LIN {X 226.123,Y -181.572,Z 120.218,A 141.236,B 90.000,C 0.000} C_DIS
LIN {X 226.096,Y -181.605,Z 120.167,A 141.228,B 90.000,C 0.000} C_DIS
LIN {X 225.969,Y -181.764,Z 120.125,A 141.188,B 90.000,C 0.000} C_DIS
LIN {X 225.915,Y -181.830,Z 120.023,A 141.171,B 90.000,C 0.000} C_DIS
LIN {X 225.787,Y -181.989,Z 119.980,A 141.130,B 90.000,C 0.000} C_DIS
LIN {X 225.761,Y -182.022,Z 119.929,A 141.122,B 90.000,C 0.000} C_DIS
LIN {X 225.721,Y -182.072,Z 119.878,A 141.109,B 90.000,C 0.000} C_DIS
LIN {X 225.528,Y -182.310,Z 119.836,A 141.049,B 90.000,C 0.000} C_DIS
LIN {X 225.488,Y -182.360,Z 119.785,A 141.036,B 90.000,C 0.000} C_DIS
LIN {X 225.462,Y -182.393,Z 119.734,A 141.028,B 90.000,C 0.000} C_DIS
LIN {X 225.333,Y -182.551,Z 119.691,A 140.988,B 90.000,C 0.000} C_DIS
LIN {X 225.306,Y -182.584,Z 119.640,A 140.979,B 90.000,C 0.000} C_DIS
LIN {X 225.266,Y -182.634,Z 119.589,A 140.967,B 90.000,C 0.000} C_DIS
LIN {X 225.073,Y -182.872,Z 119.547,A 140.906,B 90.000,C 0.000} C_DIS
LIN {X 225.033,Y -182.921,Z 119.496,A 140.894,B 90.000,C 0.000} C_DIS
LIN {X 225.006,Y -182.954,Z 119.445,A 140.885,B 90.000,C 0.000} C_DIS
LIN {X 224.877,Y -183.112,Z 119.402,A 140.845,B 90.000,C 0.000} C_DIS
LIN {X 224.824,Y -183.178,Z 119.300,A 140.828,B 90.000,C 0.000} C_DIS
LIN {X 224.695,Y -183.336,Z 119.258,A 140.788,B 90.000,C 0.000} C_DIS
LIN {X 224.668,Y -183.369,Z 119.207,A 140.779,B 90.000,C 0.000} C_DIS
LIN {X 224.628,Y -183.419,Z 119.156,A 140.767,B 90.000,C 0.000} C_DIS
LIN {X 224.434,Y -183.656,Z 119.113,A 140.706,B 90.000,C 0.000} C_DIS
LIN {X 224.394,Y -183.705,Z 119.062,A 140.694,B 90.000,C 0.000} C_DIS
LIN {X 224.367,Y -183.738,Z 119.011,A 140.685,B 90.000,C 0.000} C_DIS
LIN {X 224.237,Y -183.896,Z 118.969,A 140.645,B 90.000,C 0.000} C_DIS
LIN {X 224.183,Y -183.961,Z 118.867,A 140.628,B 90.000,C 0.000} C_DIS
LIN {X 224.054,Y -184.119,Z 118.824,A 140.588,B 90.000,C 0.000} C_DIS
LIN {X 224.027,Y -184.152,Z 118.773,A 140.580,B 90.000,C 0.000} C_DIS
LIN {X 223.986,Y -184.201,Z 118.722,A 140.567,B 90.000,C 0.000} C_DIS
LIN {X 223.792,Y -184.438,Z 118.680,A 140.506,B 90.000,C 0.000} C_DIS
LIN {X 223.751,Y -184.487,Z 118.629,A 140.494,B 90.000,C 0.000} C_DIS
LIN {X 223.724,Y -184.519,Z 118.578,A 140.485,B 90.000,C 0.000} C_DIS
LIN {X 223.594,Y -184.677,Z 118.535,A 140.445,B 90.000,C 0.000} C_DIS
LIN {X 223.567,Y -184.710,Z 118.484,A 140.437,B 90.000,C 0.000} C_DIS
LIN {X 223.527,Y -184.759,Z 118.433,A 140.424,B 90.000,C 0.000} C_DIS
LIN {X 223.332,Y -184.995,Z 118.391,A 140.364,B 90.000,C 0.000} C_DIS
LIN {X 223.291,Y -185.044,Z 118.340,A 140.351,B 90.000,C 0.000} C_DIS
LIN {X 223.264,Y -185.076,Z 118.288,A 140.343,B 90.000,C 0.000} C_DIS
LIN {X 223.134,Y -185.233,Z 118.246,A 140.302,B 90.000,C 0.000} C_DIS
LIN {X 223.079,Y -185.299,Z 118.144,A 140.286,B 90.000,C 0.000} C_DIS
LIN {X 222.949,Y -185.456,Z 118.101,A 140.245,B 90.000,C 0.000} C_DIS
LIN {X 222.922,Y -185.488,Z 118.050,A 140.237,B 90.000,C 0.000} C_DIS
LIN {X 222.881,Y -185.537,Z 117.999,A 140.224,B 90.000,C 0.000} C_DIS
LIN {X 222.685,Y -185.773,Z 117.957,A 140.164,B 90.000,C 0.000} C_DIS
LIN {X 222.644,Y -185.822,Z 117.906,A 140.151,B 90.000,C 0.000} C_DIS
LIN {X 222.617,Y -185.854,Z 117.855,A 140.143,B 90.000,C 0.000} C_DIS
LIN {X 222.486,Y -186.011,Z 117.812,A 140.102,B 90.000,C 0.000} C_DIS
LIN {X 222.459,Y -186.043,Z 117.761,A 140.094,B 90.000,C 0.000} C_DIS
LIN {X 222.418,Y -186.092,Z 117.710,A 140.082,B 90.000,C 0.000} C_DIS
LIN {X 222.221,Y -186.327,Z 117.668,A 140.021,B 90.000,C 0.000} C_DIS
LIN {X 222.180,Y -186.376,Z 117.617,A 140.008,B 90.000,C 0.000} C_DIS
LIN {X 222.153,Y -186.408,Z 117.566,A 140.000,B 90.000,C 0.000} C_DIS
LIN {X 222.022,Y -186.565,Z 117.523,A 139.960,B 90.000,C 0.000} C_DIS
LIN {X 221.967,Y -186.630,Z 117.421,A 139.943,B 90.000,C 0.000} C_DIS
LIN {X 221.836,Y -186.786,Z 117.379,A 139.903,B 90.000,C 0.000} C_DIS
LIN {X 221.808,Y -186.818,Z 117.328,A 139.894,B 90.000,C 0.000} C_DIS
LIN {X 221.767,Y -186.867,Z 117.277,A 139.882,B 90.000,C 0.000} C_DIS
LIN {X 221.570,Y -187.101,Z 117.234,A 139.821,B 90.000,C 0.000} C_DIS
LIN {X 221.529,Y -187.150,Z 117.183,A 139.809,B 90.000,C 0.000} C_DIS
LIN {X 221.501,Y -187.182,Z 117.132,A 139.800,B 90.000,C 0.000} C_DIS
LIN {X 221.370,Y -187.338,Z 117.090,A 139.760,B 90.000,C 0.000} C_DIS
LIN {X 221.315,Y -187.403,Z 116.988,A 139.743,B 90.000,C 0.000} C_DIS
LIN {X 221.183,Y -187.559,Z 116.945,A 139.703,B 90.000,C 0.000} C_DIS
LIN {X 221.155,Y -187.591,Z 116.894,A 139.694,B 90.000,C 0.000} C_DIS
LIN {X 221.114,Y -187.640,Z 116.843,A 139.682,B 90.000,C 0.000} C_DIS
LIN {X 220.916,Y -187.873,Z 116.801,A 139.621,B 90.000,C 0.000} C_DIS
LIN {X 220.875,Y -187.921,Z 116.750,A 139.609,B 90.000,C 0.000} C_DIS
LIN {X 220.847,Y -187.954,Z 116.699,A 139.600,B 90.000,C 0.000} C_DIS
LIN {X 220.715,Y -188.109,Z 116.656,A 139.560,B 90.000,C 0.000} C_DIS
LIN {X 220.687,Y -188.141,Z 116.605,A 139.552,B 90.000,C 0.000} C_DIS
LIN {X 220.646,Y -188.190,Z 116.554,A 139.539,B 90.000,C 0.000} C_DIS
LIN {X 220.447,Y -188.423,Z 116.512,A 139.478,B 90.000,C 0.000} C_DIS
LIN {X 220.406,Y -188.471,Z 116.461,A 139.466,B 90.000,C 0.000} C_DIS
LIN {X 220.378,Y -188.503,Z 116.410,A 139.457,B 90.000,C 0.000} C_DIS
LIN {X 220.245,Y -188.659,Z 116.367,A 139.417,B 90.000,C 0.000} C_DIS
LIN {X 220.218,Y -188.691,Z 116.316,A 139.409,B 90.000,C 0.000} C_DIS
LIN {X 220.176,Y -188.739,Z 116.265,A 139.396,B 90.000,C 0.000} C_DIS
LIN {X 219.977,Y -188.972,Z 116.223,A 139.336,B 90.000,C 0.000} C_DIS
LIN {X 219.935,Y -189.020,Z 116.172,A 139.323,B 90.000,C 0.000} C_DIS
LIN {X 219.908,Y -189.052,Z 116.121,A 139.315,B 90.000,C 0.000} C_DIS
LIN {X 219.774,Y -189.207,Z 116.078,A 139.274,B 90.000,C 0.000} C_DIS
LIN {X 219.719,Y -189.271,Z 115.976,A 139.258,B 90.000,C 0.000} C_DIS
LIN {X 219.586,Y -189.426,Z 115.934,A 139.217,B 90.000,C 0.000} C_DIS
LIN {X 219.558,Y -189.458,Z 115.883,A 139.209,B 90.000,C 0.000} C_DIS
LIN {X 219.516,Y -189.506,Z 115.831,A 139.196,B 90.000,C 0.000} C_DIS
LIN {X 219.316,Y -189.738,Z 115.789,A 139.136,B 90.000,C 0.000} C_DIS
LIN {X 219.274,Y -189.786,Z 115.738,A 139.123,B 90.000,C 0.000} C_DIS
LIN {X 219.247,Y -189.818,Z 115.687,A 139.115,B 90.000,C 0.000} C_DIS
LIN {X 219.113,Y -189.972,Z 115.645,A 139.075,B 90.000,C 0.000} C_DIS
LIN {X 219.057,Y -190.036,Z 115.542,A 139.058,B 90.000,C 0.000} C_DIS
LIN {X 218.924,Y -190.191,Z 115.500,A 139.017,B 90.000,C 0.000} C_DIS
LIN {X 218.896,Y -190.223,Z 115.449,A 139.009,B 90.000,C 0.000} C_DIS
LIN {X 218.854,Y -190.271,Z 115.398,A 138.996,B 90.000,C 0.000} C_DIS
LIN {X 218.653,Y -190.502,Z 115.355,A 138.936,B 90.000,C 0.000} C_DIS
LIN {X 218.611,Y -190.550,Z 115.304,A 138.923,B 90.000,C 0.000} C_DIS
LIN {X 218.583,Y -190.582,Z 115.253,A 138.915,B 90.000,C 0.000} C_DIS
LIN {X 218.449,Y -190.736,Z 115.211,A 138.875,B 90.000,C 0.000} C_DIS
LIN {X 218.421,Y -190.768,Z 115.160,A 138.866,B 90.000,C 0.000} C_DIS
LIN {X 218.379,Y -190.816,Z 115.109,A 138.854,B 90.000,C 0.000} C_DIS
LIN {X 218.178,Y -191.046,Z 115.066,A 138.793,B 90.000,C 0.000} C_DIS
LIN {X 218.136,Y -191.094,Z 115.015,A 138.781,B 90.000,C 0.000} C_DIS
LIN {X 218.108,Y -191.126,Z 114.964,A 138.772,B 90.000,C 0.000} C_DIS
LIN {X 217.973,Y -191.279,Z 114.922,A 138.732,B 90.000,C 0.000} C_DIS
LIN {X 217.917,Y -191.343,Z 114.820,A 138.715,B 90.000,C 0.000} C_DIS
LIN {X 217.782,Y -191.497,Z 114.777,A 138.675,B 90.000,C 0.000} C_DIS
LIN {X 217.754,Y -191.528,Z 114.726,A 138.666,B 90.000,C 0.000} C_DIS
LIN {X 217.712,Y -191.576,Z 114.675,A 138.654,B 90.000,C 0.000} C_DIS
LIN {X 217.510,Y -191.806,Z 114.633,A 138.593,B 90.000,C 0.000} C_DIS
LIN {X 217.468,Y -191.854,Z 114.582,A 138.581,B 90.000,C 0.000} C_DIS
LIN {X 217.439,Y -191.886,Z 114.531,A 138.572,B 90.000,C 0.000} C_DIS
LIN {X 217.304,Y -192.039,Z 114.488,A 138.532,B 90.000,C 0.000} C_DIS
LIN {X 217.248,Y -192.102,Z 114.386,A 138.515,B 90.000,C 0.000} C_DIS
LIN {X 217.113,Y -192.255,Z 114.344,A 138.475,B 90.000,C 0.000} C_DIS
LIN {X 217.085,Y -192.287,Z 114.293,A 138.466,B 90.000,C 0.000} C_DIS
LIN {X 217.042,Y -192.335,Z 114.242,A 138.454,B 90.000,C 0.000} C_DIS
LIN {X 216.839,Y -192.564,Z 114.199,A 138.393,B 90.000,C 0.000} C_DIS
LIN {X 216.797,Y -192.611,Z 114.148,A 138.381,B 90.000,C 0.000} C_DIS
LIN {X 216.769,Y -192.643,Z 114.097,A 138.372,B 90.000,C 0.000} C_DIS
LIN {X 216.633,Y -192.796,Z 114.055,A 138.332,B 90.000,C 0.000} C_DIS
LIN {X 216.605,Y -192.827,Z 114.004,A 138.324,B 90.000,C 0.000} C_DIS
LIN {X 216.563,Y -192.875,Z 113.953,A 138.311,B 90.000,C 0.000} C_DIS
LIN {X 216.359,Y -193.103,Z 113.910,A 138.251,B 90.000,C 0.000} C_DIS
LIN {X 216.316,Y -193.151,Z 113.859,A 138.238,B 90.000,C 0.000} C_DIS
LIN {X 216.288,Y -193.183,Z 113.808,A 138.230,B 90.000,C 0.000} C_DIS
LIN {X 216.152,Y -193.335,Z 113.766,A 138.189,B 90.000,C 0.000} C_DIS
LIN {X 216.095,Y -193.398,Z 113.664,A 138.173,B 90.000,C 0.000} C_DIS
LIN {X 215.959,Y -193.550,Z 113.621,A 138.132,B 90.000,C 0.000} C_DIS
LIN {X 215.931,Y -193.582,Z 113.570,A 138.124,B 90.000,C 0.000} C_DIS
LIN {X 215.888,Y -193.629,Z 113.519,A 138.111,B 90.000,C 0.000} C_DIS
LIN {X 215.684,Y -193.857,Z 113.477,A 138.051,B 90.000,C 0.000} C_DIS
LIN {X 215.641,Y -193.904,Z 113.426,A 138.038,B 90.000,C 0.000} C_DIS
LIN {X 215.613,Y -193.936,Z 113.375,A 138.030,B 90.000,C 0.000} C_DIS
LIN {X 215.476,Y -194.088,Z 113.332,A 137.989,B 90.000,C 0.000} C_DIS
LIN {X 215.448,Y -194.119,Z 113.281,A 137.981,B 90.000,C 0.000} C_DIS
LIN {X 215.405,Y -194.166,Z 113.230,A 137.968,B 90.000,C 0.000} C_DIS
LIN {X 215.200,Y -194.394,Z 113.188,A 137.908,B 90.000,C 0.000} C_DIS
LIN {X 215.157,Y -194.441,Z 113.137,A 137.895,B 90.000,C 0.000} C_DIS
LIN {X 215.129,Y -194.473,Z 113.085,A 137.887,B 90.000,C 0.000} C_DIS
LIN {X 214.992,Y -194.624,Z 113.043,A 137.847,B 90.000,C 0.000} C_DIS
LIN {X 214.935,Y -194.687,Z 112.941,A 137.830,B 90.000,C 0.000} C_DIS
LIN {X 214.798,Y -194.838,Z 112.898,A 137.790,B 90.000,C 0.000} C_DIS
LIN {X 214.769,Y -194.870,Z 112.847,A 137.781,B 90.000,C 0.000} C_DIS
LIN {X 214.726,Y -194.917,Z 112.796,A 137.769,B 90.000,C 0.000} C_DIS
LIN {X 214.521,Y -195.143,Z 112.754,A 137.708,B 90.000,C 0.000} C_DIS
LIN {X 214.478,Y -195.190,Z 112.703,A 137.695,B 90.000,C 0.000} C_DIS
LIN {X 214.449,Y -195.222,Z 112.652,A 137.687,B 90.000,C 0.000} C_DIS
LIN {X 214.312,Y -195.373,Z 112.609,A 137.647,B 90.000,C 0.000} C_DIS
LIN {X 214.254,Y -195.436,Z 112.507,A 137.630,B 90.000,C 0.000} C_DIS
LIN {X 214.117,Y -195.586,Z 112.465,A 137.590,B 90.000,C 0.000} C_DIS
LIN {X 214.088,Y -195.618,Z 112.414,A 137.581,B 90.000,C 0.000} C_DIS
LIN {X 214.045,Y -195.665,Z 112.363,A 137.569,B 90.000,C 0.000} C_DIS
LIN {X 213.838,Y -195.891,Z 112.320,A 137.508,B 90.000,C 0.000} C_DIS
LIN {X 213.795,Y -195.938,Z 112.269,A 137.496,B 90.000,C 0.000} C_DIS
LIN {X 213.767,Y -195.969,Z 112.218,A 137.487,B 90.000,C 0.000} C_DIS
LIN {X 213.629,Y -196.119,Z 112.176,A 137.447,B 90.000,C 0.000} C_DIS
LIN {X 213.600,Y -196.151,Z 112.125,A 137.439,B 90.000,C 0.000} C_DIS
LIN {X 213.557,Y -196.197,Z 112.074,A 137.426,B 90.000,C 0.000} C_DIS
LIN {X 213.350,Y -196.423,Z 112.031,A 137.365,B 90.000,C 0.000} C_DIS
LIN {X 213.307,Y -196.470,Z 111.980,A 137.353,B 90.000,C 0.000} C_DIS
LIN {X 213.278,Y -196.501,Z 111.929,A 137.344,B 90.000,C 0.000} C_DIS
LIN {X 213.139,Y -196.651,Z 111.887,A 137.304,B 90.000,C 0.000} C_DIS
LIN {X 213.111,Y -196.682,Z 111.836,A 137.296,B 90.000,C 0.000} C_DIS
LIN {X 213.067,Y -196.729,Z 111.785,A 137.283,B 90.000,C 0.000} C_DIS
LIN {X 212.860,Y -196.954,Z 111.742,A 137.223,B 90.000,C 0.000} C_DIS
LIN {X 212.816,Y -197.001,Z 111.691,A 137.210,B 90.000,C 0.000} C_DIS
LIN {X 212.787,Y -197.032,Z 111.640,A 137.202,B 90.000,C 0.000} C_DIS
LIN {X 212.649,Y -197.181,Z 111.598,A 137.161,B 90.000,C 0.000} C_DIS
LIN {X 212.591,Y -197.244,Z 111.496,A 137.145,B 90.000,C 0.000} C_DIS
LIN {X 212.452,Y -197.393,Z 111.453,A 137.104,B 90.000,C 0.000} C_DIS
LIN {X 212.423,Y -197.424,Z 111.402,A 137.096,B 90.000,C 0.000} C_DIS
LIN {X 212.380,Y -197.471,Z 111.351,A 137.083,B 90.000,C 0.000} C_DIS
LIN {X 212.171,Y -197.695,Z 111.309,A 137.023,B 90.000,C 0.000} C_DIS
LIN {X 212.128,Y -197.742,Z 111.258,A 137.010,B 90.000,C 0.000} C_DIS
LIN {X 212.099,Y -197.773,Z 111.207,A 137.002,B 90.000,C 0.000} C_DIS
LIN {X 211.959,Y -197.922,Z 111.164,A 136.961,B 90.000,C 0.000} C_DIS
LIN {X 211.902,Y -197.984,Z 111.062,A 136.945,B 90.000,C 0.000} C_DIS
LIN {X 211.762,Y -198.133,Z 111.020,A 136.904,B 90.000,C 0.000} C_DIS
LIN {X 211.733,Y -198.164,Z 110.969,A 136.896,B 90.000,C 0.000} C_DIS
LIN {X 211.690,Y -198.211,Z 110.918,A 136.883,B 90.000,C 0.000} C_DIS
LIN {X 211.480,Y -198.434,Z 110.875,A 136.823,B 90.000,C 0.000} C_DIS
LIN {X 211.437,Y -198.481,Z 110.824,A 136.810,B 90.000,C 0.000} C_DIS
LIN {X 211.408,Y -198.512,Z 110.773,A 136.802,B 90.000,C 0.000} C_DIS
LIN {X 211.268,Y -198.660,Z 110.731,A 136.762,B 90.000,C 0.000} C_DIS
LIN {X 211.239,Y -198.691,Z 110.680,A 136.753,B 90.000,C 0.000} C_DIS
LIN {X 211.195,Y -198.738,Z 110.628,A 136.741,B 90.000,C 0.000} C_DIS
LIN {X 210.985,Y -198.961,Z 110.586,A 136.680,B 90.000,C 0.000} C_DIS
LIN {X 210.941,Y -199.007,Z 110.535,A 136.668,B 90.000,C 0.000} C_DIS
LIN {X 210.912,Y -199.038,Z 110.484,A 136.659,B 90.000,C 0.000} C_DIS
LIN {X 210.772,Y -199.186,Z 110.442,A 136.619,B 90.000,C 0.000} C_DIS
LIN {X 210.714,Y -199.248,Z 110.339,A 136.602,B 90.000,C 0.000} C_DIS
LIN {X 210.573,Y -199.396,Z 110.297,A 136.562,B 90.000,C 0.000} C_DIS
LIN {X 210.544,Y -199.427,Z 110.246,A 136.553,B 90.000,C 0.000} C_DIS
LIN {X 210.500,Y -199.473,Z 110.195,A 136.541,B 90.000,C 0.000} C_DIS
LIN {X 210.290,Y -199.695,Z 110.152,A 136.480,B 90.000,C 0.000} C_DIS
LIN {X 210.246,Y -199.742,Z 110.101,A 136.468,B 90.000,C 0.000} C_DIS
LIN {X 210.217,Y -199.772,Z 110.050,A 136.459,B 90.000,C 0.000} C_DIS
LIN {X 210.076,Y -199.920,Z 110.008,A 136.419,B 90.000,C 0.000} C_DIS
LIN {X 210.017,Y -199.982,Z 109.906,A 136.402,B 90.000,C 0.000} C_DIS
LIN {X 209.877,Y -200.130,Z 109.863,A 136.362,B 90.000,C 0.000} C_DIS
LIN {X 209.847,Y -200.160,Z 109.812,A 136.353,B 90.000,C 0.000} C_DIS
LIN {X 209.803,Y -200.206,Z 109.761,A 136.341,B 90.000,C 0.000} C_DIS
LIN {X 209.592,Y -200.428,Z 109.719,A 136.280,B 90.000,C 0.000} C_DIS
LIN {X 209.548,Y -200.474,Z 109.668,A 136.268,B 90.000,C 0.000} C_DIS
LIN {X 209.518,Y -200.505,Z 109.617,A 136.259,B 90.000,C 0.000} C_DIS
LIN {X 209.377,Y -200.652,Z 109.574,A 136.219,B 90.000,C 0.000} C_DIS
LIN {X 209.348,Y -200.683,Z 109.523,A 136.211,B 90.000,C 0.000} C_DIS
LIN {X 209.304,Y -200.729,Z 109.472,A 136.198,B 90.000,C 0.000} C_DIS
LIN {X 209.092,Y -200.949,Z 109.430,A 136.138,B 90.000,C 0.000} C_DIS
LIN {X 209.048,Y -200.995,Z 109.379,A 136.125,B 90.000,C 0.000} C_DIS
LIN {X 209.018,Y -201.026,Z 109.328,A 136.117,B 90.000,C 0.000} C_DIS
LIN {X 208.877,Y -201.173,Z 109.285,A 136.076,B 90.000,C 0.000} C_DIS
LIN {X 208.818,Y -201.234,Z 109.183,A 136.059,B 90.000,C 0.000} C_DIS
LIN {X 208.676,Y -201.381,Z 109.141,A 136.019,B 90.000,C 0.000} C_DIS
LIN {X 208.646,Y -201.412,Z 109.090,A 136.011,B 90.000,C 0.000} C_DIS
LIN {X 208.602,Y -201.458,Z 109.039,A 135.998,B 90.000,C 0.000} C_DIS
LIN {X 208.389,Y -201.678,Z 108.996,A 135.938,B 90.000,C 0.000} C_DIS
LIN {X 208.345,Y -201.723,Z 108.945,A 135.925,B 90.000,C 0.000} C_DIS
LIN {X 208.316,Y -201.754,Z 108.894,A 135.917,B 90.000,C 0.000} C_DIS
LIN {X 208.173,Y -201.901,Z 108.852,A 135.876,B 90.000,C 0.000} C_DIS
LIN {X 208.144,Y -201.931,Z 108.801,A 135.868,B 90.000,C 0.000} C_DIS
LIN {X 208.100,Y -201.977,Z 108.750,A 135.855,B 90.000,C 0.000} C_DIS
LIN {X 207.886,Y -202.196,Z 108.707,A 135.795,B 90.000,C 0.000} C_DIS
LIN {X 207.842,Y -202.242,Z 108.656,A 135.782,B 90.000,C 0.000} C_DIS
LIN {X 207.812,Y -202.272,Z 108.605,A 135.774,B 90.000,C 0.000} C_DIS
LIN {X 207.670,Y -202.419,Z 108.563,A 135.734,B 90.000,C 0.000} C_DIS
LIN {X 207.610,Y -202.479,Z 108.461,A 135.717,B 90.000,C 0.000} C_DIS
LIN {X 207.468,Y -202.626,Z 108.418,A 135.677,B 90.000,C 0.000} C_DIS
LIN {X 207.438,Y -202.656,Z 108.367,A 135.668,B 90.000,C 0.000} C_DIS
LIN {X 207.394,Y -202.701,Z 108.316,A 135.656,B 90.000,C 0.000} C_DIS
LIN {X 207.179,Y -202.920,Z 108.274,A 135.595,B 90.000,C 0.000} C_DIS
LIN {X 207.135,Y -202.966,Z 108.223,A 135.582,B 90.000,C 0.000} C_DIS
LIN {X 207.105,Y -202.996,Z 108.172,A 135.574,B 90.000,C 0.000} C_DIS
LIN {X 206.962,Y -203.142,Z 108.129,A 135.534,B 90.000,C 0.000} C_DIS
LIN {X 206.933,Y -203.172,Z 108.078,A 135.525,B 90.000,C 0.000} C_DIS
LIN {X 206.888,Y -203.218,Z 108.027,A 135.513,B 90.000,C 0.000} C_DIS
LIN {X 206.673,Y -203.436,Z 107.985,A 135.452,B 90.000,C 0.000} C_DIS
LIN {X 206.629,Y -203.481,Z 107.933,A 135.440,B 90.000,C 0.000} C_DIS
LIN {X 206.599,Y -203.512,Z 107.882,A 135.431,B 90.000,C 0.000} C_DIS
LIN {X 206.455,Y -203.657,Z 107.840,A 135.391,B 90.000,C 0.000} C_DIS
LIN {X 206.396,Y -203.717,Z 107.738,A 135.374,B 90.000,C 0.000} C_DIS
LIN {X 206.252,Y -203.863,Z 107.695,A 135.334,B 90.000,C 0.000} C_DIS
LIN {X 206.222,Y -203.893,Z 107.644,A 135.325,B 90.000,C 0.000} C_DIS
LIN {X 206.178,Y -203.938,Z 107.593,A 135.313,B 90.000,C 0.000} C_DIS
LIN {X 205.962,Y -204.156,Z 107.551,A 135.252,B 90.000,C 0.000} C_DIS
LIN {X 205.917,Y -204.201,Z 107.500,A 135.240,B 90.000,C 0.000} C_DIS
LIN {X 205.887,Y -204.231,Z 107.449,A 135.231,B 90.000,C 0.000} C_DIS
LIN {X 205.744,Y -204.376,Z 107.406,A 135.191,B 90.000,C 0.000} C_DIS
LIN {X 205.684,Y -204.436,Z 107.304,A 135.174,B 90.000,C 0.000} C_DIS
LIN {X 205.540,Y -204.581,Z 107.262,A 135.134,B 90.000,C 0.000} C_DIS
LIN {X 205.510,Y -204.611,Z 107.211,A 135.126,B 90.000,C 0.000} C_DIS
LIN {X 205.465,Y -204.656,Z 107.160,A 135.113,B 90.000,C 0.000} C_DIS
LIN {X 205.249,Y -204.873,Z 107.117,A 135.052,B 90.000,C 0.000} C_DIS
LIN {X 205.204,Y -204.918,Z 107.066,A 135.040,B 90.000,C 0.000} C_DIS
LIN {X 205.174,Y -204.948,Z 107.015,A 135.032,B 90.000,C 0.000} C_DIS
LIN {X 205.029,Y -205.093,Z 106.973,A 134.991,B 90.000,C 0.000} C_DIS
LIN {X 204.999,Y -205.123,Z 106.922,A 134.983,B 90.000,C 0.000} C_DIS
LIN {X 204.954,Y -205.168,Z 106.871,A 134.970,B 90.000,C 0.000} C_DIS
LIN {X 204.738,Y -205.384,Z 106.828,A 134.910,B 90.000,C 0.000} C_DIS
LIN {X 204.692,Y -205.429,Z 106.777,A 134.897,B 90.000,C 0.000} C_DIS
LIN {X 204.662,Y -205.459,Z 106.726,A 134.889,B 90.000,C 0.000} C_DIS
LIN {X 204.518,Y -205.603,Z 106.684,A 134.848,B 90.000,C 0.000} C_DIS
LIN {X 204.458,Y -205.663,Z 106.582,A 134.832,B 90.000,C 0.000} C_DIS
LIN {X 204.313,Y -205.807,Z 106.539,A 134.791,B 90.000,C 0.000} C_DIS
LIN {X 204.283,Y -205.836,Z 106.488,A 134.783,B 90.000,C 0.000} C_DIS
LIN {X 204.237,Y -205.881,Z 106.437,A 134.770,B 90.000,C 0.000} C_DIS
LIN {X 204.020,Y -206.097,Z 106.395,A 134.710,B 90.000,C 0.000} C_DIS
LIN {X 203.975,Y -206.142,Z 106.344,A 134.697,B 90.000,C 0.000} C_DIS
LIN {X 203.944,Y -206.171,Z 106.293,A 134.689,B 90.000,C 0.000} C_DIS
LIN {X 203.799,Y -206.315,Z 106.250,A 134.649,B 90.000,C 0.000} C_DIS
LIN {X 203.769,Y -206.345,Z 106.199,A 134.640,B 90.000,C 0.000} C_DIS
LIN {X 203.724,Y -206.390,Z 106.148,A 134.628,B 90.000,C 0.000} C_DIS
LIN {X 203.506,Y -206.605,Z 106.106,A 134.567,B 90.000,C 0.000} C_DIS
LIN {X 203.460,Y -206.649,Z 106.055,A 134.554,B 90.000,C 0.000} C_DIS
LIN {X 203.430,Y -206.679,Z 106.004,A 134.546,B 90.000,C 0.000} C_DIS
LIN {X 203.284,Y -206.822,Z 105.961,A 134.506,B 90.000,C 0.000} C_DIS
LIN {X 203.224,Y -206.882,Z 105.859,A 134.489,B 90.000,C 0.000} C_DIS
LIN {X 203.078,Y -207.025,Z 105.817,A 134.449,B 90.000,C 0.000} C_DIS
LIN {X 203.048,Y -207.054,Z 105.766,A 134.440,B 90.000,C 0.000} C_DIS
LIN {X 203.002,Y -207.099,Z 105.715,A 134.428,B 90.000,C 0.000} C_DIS
LIN {X 202.784,Y -207.313,Z 105.672,A 134.367,B 90.000,C 0.000} C_DIS
LIN {X 202.738,Y -207.358,Z 105.621,A 134.355,B 90.000,C 0.000} C_DIS
LIN {X 202.708,Y -207.387,Z 105.570,A 134.346,B 90.000,C 0.000} C_DIS
LIN {X 202.562,Y -207.530,Z 105.528,A 134.306,B 90.000,C 0.000} C_DIS
LIN {X 202.531,Y -207.560,Z 105.477,A 134.297,B 90.000,C 0.000} C_DIS
LIN {X 202.486,Y -207.604,Z 105.425,A 134.285,B 90.000,C 0.000} C_DIS
LIN {X 202.266,Y -207.818,Z 105.383,A 134.224,B 90.000,C 0.000} C_DIS
LIN {X 202.221,Y -207.862,Z 105.332,A 134.212,B 90.000,C 0.000} C_DIS
LIN {X 202.190,Y -207.892,Z 105.281,A 134.203,B 90.000,C 0.000} C_DIS
LIN {X 202.044,Y -208.034,Z 105.238,A 134.163,B 90.000,C 0.000} C_DIS
LIN {X 201.983,Y -208.093,Z 105.136,A 134.146,B 90.000,C 0.000} C_DIS
LIN {X 201.836,Y -208.236,Z 105.094,A 134.106,B 90.000,C 0.000} C_DIS
LIN {X 201.806,Y -208.265,Z 105.043,A 134.098,B 90.000,C 0.000} C_DIS
LIN {X 201.760,Y -208.309,Z 104.992,A 134.085,B 90.000,C 0.000} C_DIS
LIN {X 201.540,Y -208.522,Z 104.949,A 134.025,B 90.000,C 0.000} C_DIS
LIN {X 201.494,Y -208.567,Z 104.898,A 134.012,B 90.000,C 0.000} C_DIS
LIN {X 201.464,Y -208.596,Z 104.847,A 134.004,B 90.000,C 0.000} C_DIS
LIN {X 201.317,Y -208.738,Z 104.805,A 133.963,B 90.000,C 0.000} C_DIS
LIN {X 201.286,Y -208.767,Z 104.754,A 133.955,B 90.000,C 0.000} C_DIS
LIN {X 201.241,Y -208.811,Z 104.703,A 133.942,B 90.000,C 0.000} C_DIS
LIN {X 201.020,Y -209.024,Z 104.660,A 133.882,B 90.000,C 0.000} C_DIS
LIN {X 200.974,Y -209.068,Z 104.609,A 133.869,B 90.000,C 0.000} C_DIS
LIN {X 200.943,Y -209.097,Z 104.558,A 133.861,B 90.000,C 0.000} C_DIS
LIN {X 200.796,Y -209.239,Z 104.516,A 133.820,B 90.000,C 0.000} C_DIS
LIN {X 200.735,Y -209.298,Z 104.414,A 133.804,B 90.000,C 0.000} C_DIS
LIN {X 200.588,Y -209.439,Z 104.371,A 133.763,B 90.000,C 0.000} C_DIS
LIN {X 200.557,Y -209.468,Z 104.320,A 133.755,B 90.000,C 0.000} C_DIS
LIN {X 200.511,Y -209.512,Z 104.269,A 133.742,B 90.000,C 0.000} C_DIS
LIN {X 200.290,Y -209.724,Z 104.227,A 133.682,B 90.000,C 0.000} C_DIS
LIN {X 200.243,Y -209.768,Z 104.176,A 133.669,B 90.000,C 0.000} C_DIS
LIN {X 200.213,Y -209.797,Z 104.125,A 133.661,B 90.000,C 0.000} C_DIS
LIN {X 200.065,Y -209.938,Z 104.082,A 133.621,B 90.000,C 0.000} C_DIS
LIN {X 200.004,Y -209.997,Z 103.980,A 133.604,B 90.000,C 0.000} C_DIS
LIN {X 199.856,Y -210.137,Z 103.938,A 133.563,B 90.000,C 0.000} C_DIS
LIN {X 199.825,Y -210.167,Z 103.887,A 133.555,B 90.000,C 0.000} C_DIS
LIN {X 199.779,Y -210.210,Z 103.836,A 133.542,B 90.000,C 0.000} C_DIS
LIN {X 199.557,Y -210.421,Z 103.793,A 133.482,B 90.000,C 0.000} C_DIS
LIN {X 199.510,Y -210.465,Z 103.742,A 133.469,B 90.000,C 0.000} C_DIS
LIN {X 199.480,Y -210.494,Z 103.691,A 133.461,B 90.000,C 0.000} C_DIS
LIN {X 199.331,Y -210.635,Z 103.649,A 133.421,B 90.000,C 0.000} C_DIS
LIN {X 199.301,Y -210.664,Z 103.598,A 133.412,B 90.000,C 0.000} C_DIS
LIN {X 199.254,Y -210.708,Z 103.547,A 133.400,B 90.000,C 0.000} C_DIS
LIN {X 199.032,Y -210.918,Z 103.504,A 133.339,B 90.000,C 0.000} C_DIS
LIN {X 198.985,Y -210.962,Z 103.453,A 133.327,B 90.000,C 0.000} C_DIS
LIN {X 198.955,Y -210.991,Z 103.402,A 133.318,B 90.000,C 0.000} C_DIS
LIN {X 198.806,Y -211.131,Z 103.360,A 133.278,B 90.000,C 0.000} C_DIS
LIN {X 198.744,Y -211.189,Z 103.258,A 133.261,B 90.000,C 0.000} C_DIS
LIN {X 198.595,Y -211.329,Z 103.215,A 133.221,B 90.000,C 0.000} C_DIS
LIN {X 198.564,Y -211.358,Z 103.164,A 133.212,B 90.000,C 0.000} C_DIS
LIN {X 198.518,Y -211.401,Z 103.113,A 133.200,B 90.000,C 0.000} C_DIS
LIN {X 198.295,Y -211.611,Z 103.071,A 133.139,B 90.000,C 0.000} C_DIS
LIN {X 198.248,Y -211.655,Z 103.020,A 133.127,B 90.000,C 0.000} C_DIS
LIN {X 198.217,Y -211.684,Z 102.968,A 133.118,B 90.000,C 0.000} C_DIS
LIN {X 198.068,Y -211.823,Z 102.926,A 133.078,B 90.000,C 0.000} C_DIS
LIN {X 198.037,Y -211.852,Z 102.875,A 133.070,B 90.000,C 0.000} C_DIS
LIN {X 197.991,Y -211.896,Z 102.824,A 133.057,B 90.000,C 0.000} C_DIS
LIN {X 197.767,Y -212.104,Z 102.782,A 132.997,B 90.000,C 0.000} C_DIS
LIN {X 197.720,Y -212.148,Z 102.730,A 132.984,B 90.000,C 0.000} C_DIS
LIN {X 197.689,Y -212.177,Z 102.679,A 132.976,B 90.000,C 0.000} C_DIS
LIN {X 197.540,Y -212.316,Z 102.637,A 132.935,B 90.000,C 0.000} C_DIS
LIN {X 197.478,Y -212.374,Z 102.535,A 132.918,B 90.000,C 0.000} C_DIS
LIN {X 197.328,Y -212.513,Z 102.492,A 132.878,B 90.000,C 0.000} C_DIS
LIN {X 197.297,Y -212.542,Z 102.441,A 132.870,B 90.000,C 0.000} C_DIS
LIN {X 197.273,Y -212.564,Z 102.390,A 132.863,B 90.000,C 0.000} C_DIS
LIN {X 197.215,Y -212.618,Z 102.369,A 132.848,B 90.000,C 0.000} C_DIS
LIN {X 197.119,Y -212.707,Z 102.317,A 132.822,B 90.000,C 0.000} C_DIS
LIN {X 197.003,Y -212.814,Z 102.192,A 132.791,B 90.000,C 0.000} C_DIS
LIN {X 196.873,Y -212.935,Z 102.014,A 132.756,B 90.000,C 0.000} C_DIS
LIN {X 196.882,Y -212.926,Z 99.514,A 132.758,B 90.000,C 0.000} C_DIS
LIN {X 196.887,Y -212.922,Z 99.055,A 132.759,B 90.000,C 0.000} C_DIS
LIN {X 196.965,Y -212.849,Z 98.268,A 132.780,B 90.000,C 0.000} C_DIS
LIN {X 196.993,Y -212.823,Z 96.353,A 132.788,B 90.000,C 0.000} C_DIS
LIN {X 197.032,Y -212.787,Z 96.010,A 132.798,B 90.000,C 0.000} C_DIS
LIN {X 197.069,Y -212.753,Z 95.977,A 132.808,B 90.000,C 0.000} C_DIS
LIN {X 197.085,Y -212.738,Z 95.898,A 132.813,B 90.000,C 0.000} C_DIS
LIN {X 197.123,Y -212.703,Z 95.767,A 132.823,B 90.000,C 0.000} C_DIS
LIN {X 197.215,Y -212.618,Z 95.609,A 132.848,B 90.000,C 0.000} C_DIS
LIN {X 197.368,Y -212.475,Z 95.469,A 132.889,B 90.000,C 0.000} C_DIS
LIN {X 197.586,Y -212.273,Z 95.432,A 132.948,B 90.000,C 0.000} C_DIS
LIN {X 197.755,Y -212.115,Z 95.453,A 132.993,B 90.000,C 0.000} C_DIS
LIN {X 197.826,Y -212.049,Z 95.504,A 133.013,B 90.000,C 0.000} C_DIS
LIN {X 197.872,Y -212.006,Z 95.555,A 133.025,B 90.000,C 0.000} C_DIS
LIN {X 198.096,Y -211.797,Z 95.597,A 133.086,B 90.000,C 0.000} C_DIS
LIN {X 198.189,Y -211.710,Z 95.700,A 133.111,B 90.000,C 0.000} C_DIS
LIN {X 198.413,Y -211.500,Z 95.742,A 133.171,B 90.000,C 0.000} C_DIS
LIN {X 198.459,Y -211.457,Z 95.793,A 133.184,B 90.000,C 0.000} C_DIS
LIN {X 198.490,Y -211.428,Z 95.844,A 133.192,B 90.000,C 0.000} C_DIS
LIN {X 198.639,Y -211.288,Z 95.887,A 133.233,B 90.000,C 0.000} C_DIS
LIN {X 198.701,Y -211.230,Z 95.989,A 133.249,B 90.000,C 0.000} C_DIS
LIN {X 198.775,Y -211.160,Z 96.010,A 133.270,B 90.000,C 0.000} C_DIS
LIN {X 198.849,Y -211.090,Z 95.989,A 133.290,B 90.000,C 0.000} C_DIS
LIN {X 198.880,Y -211.061,Z 95.938,A 133.298,B 90.000,C 0.000} C_DIS
LIN {X 198.849,Y -211.090,Z 95.887,A 133.290,B 90.000,C 0.000} C_DIS
LIN {X 198.701,Y -211.230,Z 95.844,A 133.249,B 90.000,C 0.000} C_DIS
LIN {X 198.639,Y -211.288,Z 95.742,A 133.233,B 90.000,C 0.000} C_DIS
LIN {X 198.490,Y -211.428,Z 95.700,A 133.192,B 90.000,C 0.000} C_DIS
LIN {X 198.428,Y -211.486,Z 95.597,A 133.175,B 90.000,C 0.000} C_DIS
LIN {X 198.279,Y -211.626,Z 95.555,A 133.135,B 90.000,C 0.000} C_DIS
LIN {X 198.217,Y -211.684,Z 95.453,A 133.118,B 90.000,C 0.000} C_DIS
LIN {X 198.068,Y -211.823,Z 95.411,A 133.078,B 90.000,C 0.000} C_DIS
LIN {X 198.006,Y -211.881,Z 95.308,A 133.061,B 90.000,C 0.000} C_DIS
LIN {X 197.857,Y -212.020,Z 95.266,A 133.021,B 90.000,C 0.000} C_DIS
LIN {X 197.795,Y -212.078,Z 95.164,A 133.004,B 90.000,C 0.000} C_DIS
LIN {X 197.645,Y -212.217,Z 95.121,A 132.964,B 90.000,C 0.000} C_DIS
LIN {X 197.614,Y -212.246,Z 95.070,A 132.955,B 90.000,C 0.000} C_DIS
LIN {X 197.568,Y -212.290,Z 95.019,A 132.943,B 90.000,C 0.000} C_DIS
LIN {X 197.344,Y -212.498,Z 94.977,A 132.882,B 90.000,C 0.000} C_DIS
LIN {X 197.297,Y -212.542,Z 94.926,A 132.870,B 90.000,C 0.000} C_DIS
LIN {X 197.266,Y -212.571,Z 94.875,A 132.861,B 90.000,C 0.000} C_DIS
LIN {X 197.116,Y -212.709,Z 94.832,A 132.821,B 90.000,C 0.000} C_DIS
LIN {X 197.054,Y -212.767,Z 94.730,A 132.804,B 90.000,C 0.000} C_DIS
LIN {X 196.904,Y -212.906,Z 94.688,A 132.764,B 90.000,C 0.000} C_DIS
LIN {X 196.842,Y -212.963,Z 94.586,A 132.747,B 90.000,C 0.000} C_DIS
LIN {X 196.692,Y -213.102,Z 94.543,A 132.707,B 90.000,C 0.000} C_DIS
LIN {X 196.629,Y -213.159,Z 94.441,A 132.690,B 90.000,C 0.000} C_DIS
LIN {X 196.479,Y -213.298,Z 94.399,A 132.650,B 90.000,C 0.000} C_DIS
LIN {X 196.420,Y -213.352,Z 94.297,A 132.634,B 90.000,C 0.000} C_DIS
LIN {X 196.353,Y -213.414,Z 94.276,A 132.616,B 90.000,C 0.000} C_DIS
LIN {X 196.264,Y -213.496,Z 94.233,A 132.592,B 90.000,C 0.000} C_DIS
LIN {X 196.182,Y -213.571,Z 94.131,A 132.570,B 90.000,C 0.000} C_DIS
LIN {X 196.035,Y -213.706,Z 93.986,A 132.531,B 90.000,C 0.000} C_DIS
LIN {X 195.928,Y -213.804,Z 93.911,A 132.502,B 90.000,C 0.000} C_DIS
LIN {X 195.782,Y -213.938,Z 93.735,A 132.463,B 90.000,C 0.000} C_DIS
LIN {X 195.652,Y -214.057,Z 93.536,A 132.428,B 90.000,C 0.000} C_DIS
LIN {X 195.596,Y -214.108,Z 93.391,A 132.413,B 90.000,C 0.000} C_DIS
LIN {X 195.412,Y -214.276,Z 93.060,A 132.364,B 90.000,C 0.000} C_DIS
LIN {X 195.367,Y -214.317,Z 92.745,A 132.352,B 90.000,C 0.000} C_DIS
LIN {X 195.329,Y -214.352,Z 92.686,A 132.341,B 90.000,C 0.000} C_DIS
LIN {X 195.290,Y -214.387,Z 92.523,A 132.331,B 90.000,C 0.000} C_DIS
LIN {X 195.290,Y -214.387,Z 91.692,A 132.331,B 90.000,C 0.000} C_DIS
LIN {X 193.944,Y -212.908,Z 91.692,A 132.331,B 90.000,C 0.000} C_DIS
WAIT SEC 0.1
RET=EKI_SetBool("oxy","torchState",FALSE)
RET = EKI_Send("oxy","torchState")
LIN {X 181.822,Y -199.601,Z 91.692,A 132.331,B 90.000,C 0.000} C_DIS
LIN {X 261.298,Y 67.997,Z 119.452,A -165.414,B 90.000,C 0.000} C_DIS
LIN {X 278.717,Y 72.530,Z 119.452,A -165.414,B 90.000,C 0.000} C_DIS
LIN {X 280.653,Y 73.033,Z 119.452,A -165.414,B 90.000,C 0.000} C_DIS
WAIT SEC 1
RET=EKI_SetBool("oxy","torchState",TRUE)
RET = EKI_Send("oxy","torchState")
LIN {X 280.533,Y 73.492,Z 116.997,A -165.320,B 90.000,C 0.000} C_DIS
LIN {X 280.464,Y 73.755,Z 115.809,A -165.266,B 90.000,C 0.000} C_DIS
LIN {X 280.445,Y 73.829,Z 113.310,A -165.251,B 90.000,C 0.000} C_DIS
LIN {X 280.463,Y 73.759,Z 112.076,A -165.266,B 90.000,C 0.000} C_DIS
LIN {X 280.438,Y 73.856,Z 112.058,A -165.246,B 90.000,C 0.000} C_DIS
LIN {X 280.408,Y 73.968,Z 112.262,A -165.223,B 90.000,C 0.000} C_DIS
LIN {X 280.334,Y 74.249,Z 112.729,A -165.165,B 90.000,C 0.000} C_DIS
LIN {X 280.271,Y 74.485,Z 113.355,A -165.117,B 90.000,C 0.000} C_DIS
LIN {X 280.251,Y 74.563,Z 114.265,A -165.101,B 90.000,C 0.000} C_DIS
LIN {X 280.231,Y 74.637,Z 116.764,A -165.086,B 90.000,C 0.000} C_DIS
LIN {X 280.220,Y 74.678,Z 117.551,A -165.078,B 90.000,C 0.000} C_DIS
LIN {X 280.162,Y 74.896,Z 119.025,A -165.033,B 90.000,C 0.000} C_DIS
LIN {X 280.001,Y 75.495,Z 121.447,A -164.911,B 90.000,C 0.000} C_DIS
LIN {X 279.930,Y 75.759,Z 122.515,A -164.857,B 90.000,C 0.000} C_DIS
LIN {X 279.907,Y 75.843,Z 122.699,A -164.839,B 90.000,C 0.000} C_DIS
LIN {X 279.823,Y 76.151,Z 123.781,A -164.776,B 90.000,C 0.000} C_DIS
LIN {X 279.812,Y 76.193,Z 123.824,A -164.768,B 90.000,C 0.000} C_DIS
LIN {X 279.788,Y 76.282,Z 124.009,A -164.749,B 90.000,C 0.000} C_DIS
LIN {X 279.690,Y 76.638,Z 125.031,A -164.676,B 90.000,C 0.000} C_DIS
LIN {X 279.586,Y 77.017,Z 125.929,A -164.599,B 90.000,C 0.000} C_DIS
LIN {X 279.570,Y 77.075,Z 126.010,A -164.587,B 90.000,C 0.000} C_DIS
LIN {X 279.550,Y 77.148,Z 126.167,A -164.572,B 90.000,C 0.000} C_DIS
LIN {X 279.525,Y 77.237,Z 126.299,A -164.554,B 90.000,C 0.000} C_DIS
LIN {X 279.490,Y 77.366,Z 126.697,A -164.527,B 90.000,C 0.000} C_DIS
LIN {X 279.433,Y 77.569,Z 127.099,A -164.486,B 90.000,C 0.000} C_DIS
LIN {X 279.417,Y 77.627,Z 127.181,A -164.474,B 90.000,C 0.000} C_DIS
LIN {X 279.410,Y 77.655,Z 127.231,A -164.468,B 90.000,C 0.000} C_DIS
LIN {X 279.388,Y 77.734,Z 127.311,A -164.452,B 90.000,C 0.000} C_DIS
LIN {X 279.349,Y 77.872,Z 127.292,A -164.424,B 90.000,C 0.000} C_DIS
LIN {X 279.373,Y 77.787,Z 126.953,A -164.441,B 90.000,C 0.000} C_DIS
LIN {X 279.377,Y 77.772,Z 126.839,A -164.444,B 90.000,C 0.000} C_DIS
LIN {X 279.429,Y 77.585,Z 126.214,A -164.482,B 90.000,C 0.000} C_DIS
LIN {X 279.577,Y 77.049,Z 123.879,A -164.592,B 90.000,C 0.000} C_DIS
LIN {X 279.586,Y 77.017,Z 123.824,A -164.599,B 90.000,C 0.000} C_DIS
LIN {X 279.596,Y 76.982,Z 123.710,A -164.606,B 90.000,C 0.000} C_DIS
LIN {X 279.605,Y 76.950,Z 123.426,A -164.613,B 90.000,C 0.000} C_DIS
LIN {X 279.614,Y 76.914,Z 123.312,A -164.620,B 90.000,C 0.000} C_DIS
LIN {X 279.624,Y 76.880,Z 123.260,A -164.627,B 90.000,C 0.000} C_DIS
LIN {X 279.654,Y 76.770,Z 122.305,A -164.649,B 90.000,C 0.000} C_DIS
LIN {X 279.661,Y 76.743,Z 122.231,A -164.655,B 90.000,C 0.000} C_DIS
LIN {X 279.670,Y 76.711,Z 121.946,A -164.662,B 90.000,C 0.000} C_DIS
LIN {X 279.685,Y 76.656,Z 121.818,A -164.673,B 90.000,C 0.000} C_DIS
LIN {X 279.715,Y 76.546,Z 120.908,A -164.695,B 90.000,C 0.000} C_DIS
LIN {X 279.748,Y 76.427,Z 118.411,A -164.720,B 90.000,C 0.000} C_DIS
LIN {X 279.744,Y 76.440,Z 115.911,A -164.717,B 90.000,C 0.000} C_DIS
LIN {X 279.687,Y 76.649,Z 113.421,A -164.674,B 90.000,C 0.000} C_DIS
LIN {X 279.559,Y 77.114,Z 110.968,A -164.579,B 90.000,C 0.000} C_DIS
LIN {X 279.367,Y 77.808,Z 108.574,A -164.437,B 90.000,C 0.000} C_DIS
LIN {X 279.103,Y 78.749,Z 106.273,A -164.244,B 90.000,C 0.000} C_DIS
LIN {X 278.816,Y 79.759,Z 104.336,A -164.036,B 90.000,C 0.000} C_DIS
LIN {X 278.465,Y 80.978,Z 102.526,A -163.785,B 90.000,C 0.000} C_DIS
LIN {X 278.438,Y 81.070,Z 102.431,A -163.767,B 90.000,C 0.000} C_DIS
LIN {X 278.358,Y 81.344,Z 101.988,A -163.710,B 90.000,C 0.000} C_DIS
LIN {X 278.342,Y 81.399,Z 101.947,A -163.699,B 90.000,C 0.000} C_DIS
LIN {X 278.326,Y 81.454,Z 101.928,A -163.688,B 90.000,C 0.000} C_DIS
LIN {X 278.117,Y 82.163,Z 101.001,A -163.541,B 90.000,C 0.000} C_DIS
LIN {X 278.102,Y 82.214,Z 100.978,A -163.531,B 90.000,C 0.000} C_DIS
LIN {X 278.077,Y 82.299,Z 100.896,A -163.513,B 90.000,C 0.000} C_DIS
LIN {X 278.028,Y 82.464,Z 100.666,A -163.480,B 90.000,C 0.000} C_DIS
LIN {X 277.768,Y 83.335,Z 99.531,A -163.300,B 90.000,C 0.000} C_DIS
LIN {X 277.727,Y 83.472,Z 99.389,A -163.272,B 90.000,C 0.000} C_DIS
LIN {X 277.678,Y 83.635,Z 99.165,A -163.238,B 90.000,C 0.000} C_DIS
LIN {X 277.558,Y 84.033,Z 98.544,A -163.156,B 90.000,C 0.000} C_DIS
LIN {X 277.530,Y 84.124,Z 98.448,A -163.137,B 90.000,C 0.000} C_DIS
LIN {X 277.513,Y 84.180,Z 98.372,A -163.126,B 90.000,C 0.000} C_DIS
LIN {X 277.426,Y 84.467,Z 97.839,A -163.066,B 90.000,C 0.000} C_DIS
LIN {X 277.055,Y 85.677,Z 95.684,A -162.816,B 90.000,C 0.000} C_DIS
LIN {X 276.745,Y 86.674,Z 93.412,A -162.610,B 90.000,C 0.000} C_DIS
LIN {X 276.493,Y 87.473,Z 91.057,A -162.444,B 90.000,C 0.000} C_DIS
LIN {X 276.298,Y 88.088,Z 88.642,A -162.317,B 90.000,C 0.000} C_DIS
LIN {X 276.200,Y 88.394,Z 86.975,A -162.253,B 90.000,C 0.000} C_DIS
LIN {X 276.099,Y 88.710,Z 84.498,A -162.188,B 90.000,C 0.000} C_DIS
LIN {X 276.059,Y 88.833,Z 82.001,A -162.162,B 90.000,C 0.000} C_DIS
LIN {X 276.055,Y 88.845,Z 79.501,A -162.160,B 90.000,C 0.000} C_DIS
LIN {X 276.092,Y 88.732,Z 77.183,A -162.183,B 90.000,C 0.000} C_DIS
LIN {X 276.146,Y 88.563,Z 75.690,A -162.218,B 90.000,C 0.000} C_DIS
LIN {X 276.163,Y 88.510,Z 75.458,A -162.229,B 90.000,C 0.000} C_DIS
LIN {X 276.166,Y 88.502,Z 75.330,A -162.231,B 90.000,C 0.000} C_DIS
LIN {X 276.135,Y 88.597,Z 75.249,A -162.211,B 90.000,C 0.000} C_DIS
LIN {X 276.066,Y 88.810,Z 75.747,A -162.167,B 90.000,C 0.000} C_DIS
LIN {X 276.062,Y 88.823,Z 75.804,A -162.164,B 90.000,C 0.000} C_DIS
LIN {X 276.056,Y 88.843,Z 75.861,A -162.160,B 90.000,C 0.000} C_DIS
LIN {X 275.931,Y 89.229,Z 76.836,A -162.080,B 90.000,C 0.000} C_DIS
LIN {X 275.904,Y 89.313,Z 76.995,A -162.063,B 90.000,C 0.000} C_DIS
LIN {X 275.897,Y 89.337,Z 77.083,A -162.058,B 90.000,C 0.000} C_DIS
LIN {X 275.823,Y 89.564,Z 77.624,A -162.011,B 90.000,C 0.000} C_DIS
LIN {X 275.817,Y 89.581,Z 77.681,A -162.007,B 90.000,C 0.000} C_DIS
LIN {X 275.808,Y 89.611,Z 77.738,A -162.001,B 90.000,C 0.000} C_DIS
LIN {X 275.796,Y 89.647,Z 77.852,A -161.993,B 90.000,C 0.000} C_DIS
LIN {X 275.791,Y 89.662,Z 77.966,A -161.990,B 90.000,C 0.000} C_DIS
LIN {X 275.716,Y 89.892,Z 78.535,A -161.942,B 90.000,C 0.000} C_DIS
LIN {X 275.708,Y 89.918,Z 78.648,A -161.937,B 90.000,C 0.000} C_DIS
LIN {X 275.603,Y 90.240,Z 79.482,A -161.870,B 90.000,C 0.000} C_DIS
LIN {X 275.599,Y 90.250,Z 79.582,A -161.868,B 90.000,C 0.000} C_DIS
LIN {X 275.505,Y 90.536,Z 80.355,A -161.809,B 90.000,C 0.000} C_DIS
LIN {X 275.485,Y 90.599,Z 80.716,A -161.795,B 90.000,C 0.000} C_DIS
LIN {X 275.474,Y 90.633,Z 80.754,A -161.788,B 90.000,C 0.000} C_DIS
LIN {X 275.460,Y 90.674,Z 80.867,A -161.780,B 90.000,C 0.000} C_DIS
LIN {X 275.456,Y 90.686,Z 80.981,A -161.777,B 90.000,C 0.000} C_DIS
LIN {X 275.329,Y 91.070,Z 82.176,A -161.698,B 90.000,C 0.000} C_DIS
LIN {X 275.325,Y 91.083,Z 82.290,A -161.695,B 90.000,C 0.000} C_DIS
LIN {X 275.294,Y 91.178,Z 82.631,A -161.675,B 90.000,C 0.000} C_DIS
LIN {X 275.180,Y 91.520,Z 83.940,A -161.604,B 90.000,C 0.000} C_DIS
LIN {X 275.098,Y 91.767,Z 85.191,A -161.552,B 90.000,C 0.000} C_DIS
LIN {X 275.087,Y 91.800,Z 85.242,A -161.545,B 90.000,C 0.000} C_DIS
LIN {X 275.016,Y 92.011,Z 86.617,A -161.502,B 90.000,C 0.000} C_DIS
LIN {X 275.007,Y 92.040,Z 86.671,A -161.495,B 90.000,C 0.000} C_DIS
LIN {X 274.997,Y 92.069,Z 86.778,A -161.490,B 90.000,C 0.000} C_DIS
LIN {X 274.915,Y 92.314,Z 89.264,A -161.438,B 90.000,C 0.000} C_DIS
LIN {X 274.894,Y 92.375,Z 90.312,A -161.426,B 90.000,C 0.000} C_DIS
LIN {X 274.889,Y 92.390,Z 90.383,A -161.423,B 90.000,C 0.000} C_DIS
LIN {X 274.896,Y 92.370,Z 90.767,A -161.427,B 90.000,C 0.000} C_DIS
LIN {X 274.889,Y 92.391,Z 90.823,A -161.422,B 90.000,C 0.000} C_DIS
LIN {X 274.939,Y 92.242,Z 93.318,A -161.453,B 90.000,C 0.000} C_DIS
LIN {X 275.068,Y 91.857,Z 95.784,A -161.534,B 90.000,C 0.000} C_DIS
LIN {X 275.286,Y 91.201,Z 98.187,A -161.670,B 90.000,C 0.000} C_DIS
LIN {X 275.563,Y 90.360,Z 100.525,A -161.845,B 90.000,C 0.000} C_DIS
LIN {X 275.888,Y 89.365,Z 102.795,A -162.052,B 90.000,C 0.000} C_DIS
LIN {X 276.213,Y 88.355,Z 105.058,A -162.262,B 90.000,C 0.000} C_DIS
LIN {X 276.513,Y 87.411,Z 107.354,A -162.457,B 90.000,C 0.000} C_DIS
LIN {X 276.743,Y 86.679,Z 109.733,A -162.609,B 90.000,C 0.000} C_DIS
LIN {X 276.887,Y 86.218,Z 112.186,A -162.704,B 90.000,C 0.000} C_DIS
LIN {X 276.949,Y 86.019,Z 114.677,A -162.746,B 90.000,C 0.000} C_DIS
LIN {X 276.971,Y 85.949,Z 115.288,A -162.760,B 90.000,C 0.000} C_DIS
LIN {X 276.965,Y 85.967,Z 115.346,A -162.756,B 90.000,C 0.000} C_DIS
LIN {X 276.977,Y 85.930,Z 116.427,A -162.764,B 90.000,C 0.000} C_DIS
LIN {X 276.973,Y 85.940,Z 116.497,A -162.762,B 90.000,C 0.000} C_DIS
LIN {X 276.989,Y 85.891,Z 118.997,A -162.772,B 90.000,C 0.000} C_DIS
LIN {X 276.984,Y 85.905,Z 121.497,A -162.769,B 90.000,C 0.000} C_DIS
LIN {X 276.980,Y 85.919,Z 123.996,A -162.766,B 90.000,C 0.000} C_DIS
LIN {X 276.945,Y 86.032,Z 126.494,A -162.743,B 90.000,C 0.000} C_DIS
LIN {X 276.881,Y 86.238,Z 128.674,A -162.700,B 90.000,C 0.000} C_DIS
LIN {X 276.823,Y 86.423,Z 130.651,A -162.662,B 90.000,C 0.000} C_DIS
LIN {X 276.825,Y 86.416,Z 130.933,A -162.663,B 90.000,C 0.000} C_DIS
LIN {X 276.869,Y 86.276,Z 130.917,A -162.692,B 90.000,C 0.000} C_DIS
LIN {X 276.921,Y 86.107,Z 130.845,A -162.727,B 90.000,C 0.000} C_DIS
LIN {X 277.048,Y 85.700,Z 130.837,A -162.811,B 90.000,C 0.000} C_DIS
LIN {X 277.223,Y 85.132,Z 130.900,A -162.929,B 90.000,C 0.000} C_DIS
LIN {X 277.341,Y 84.747,Z 131.079,A -163.008,B 90.000,C 0.000} C_DIS
LIN {X 277.371,Y 84.649,Z 131.452,A -163.029,B 90.000,C 0.000} C_DIS
LIN {X 277.444,Y 84.410,Z 133.939,A -163.078,B 90.000,C 0.000} C_DIS
LIN {X 277.488,Y 84.263,Z 136.396,A -163.108,B 90.000,C 0.000} C_DIS
LIN {X 277.483,Y 84.282,Z 136.455,A -163.104,B 90.000,C 0.000} C_DIS
LIN {X 277.485,Y 84.275,Z 137.730,A -163.106,B 90.000,C 0.000} C_DIS
LIN {X 277.442,Y 84.414,Z 140.226,A -163.077,B 90.000,C 0.000} C_DIS
LIN {X 277.408,Y 84.526,Z 141.334,A -163.054,B 90.000,C 0.000} C_DIS
LIN {X 277.392,Y 84.581,Z 141.462,A -163.043,B 90.000,C 0.000} C_DIS
LIN {X 277.272,Y 84.973,Z 143.928,A -162.962,B 90.000,C 0.000} C_DIS
LIN {X 277.225,Y 85.127,Z 144.690,A -162.930,B 90.000,C 0.000} C_DIS
LIN {X 277.199,Y 85.209,Z 144.918,A -162.913,B 90.000,C 0.000} C_DIS
LIN {X 277.193,Y 85.230,Z 145.103,A -162.909,B 90.000,C 0.000} C_DIS
LIN {X 277.047,Y 85.703,Z 146.741,A -162.811,B 90.000,C 0.000} C_DIS
LIN {X 277.042,Y 85.718,Z 146.869,A -162.808,B 90.000,C 0.000} C_DIS
LIN {X 277.032,Y 85.751,Z 146.981,A -162.801,B 90.000,C 0.000} C_DIS
LIN {X 277.016,Y 85.803,Z 147.023,A -162.790,B 90.000,C 0.000} C_DIS
LIN {X 277.008,Y 85.827,Z 147.151,A -162.785,B 90.000,C 0.000} C_DIS
LIN {X 276.909,Y 86.147,Z 148.084,A -162.719,B 90.000,C 0.000} C_DIS
LIN {X 276.896,Y 86.189,Z 148.289,A -162.710,B 90.000,C 0.000} C_DIS
LIN {X 276.602,Y 87.127,Z 150.451,A -162.516,B 90.000,C 0.000} C_DIS
LIN {X 276.592,Y 87.160,Z 150.565,A -162.509,B 90.000,C 0.000} C_DIS
LIN {X 276.538,Y 87.331,Z 150.963,A -162.474,B 90.000,C 0.000} C_DIS
LIN {X 276.151,Y 88.547,Z 153.112,A -162.222,B 90.000,C 0.000} C_DIS
LIN {X 275.791,Y 89.662,Z 154.777,A -161.990,B 90.000,C 0.000} C_DIS
LIN {X 275.770,Y 89.725,Z 154.832,A -161.977,B 90.000,C 0.000} C_DIS
LIN {X 275.761,Y 89.753,Z 154.869,A -161.971,B 90.000,C 0.000} C_DIS
LIN {X 275.729,Y 89.852,Z 155.037,A -161.951,B 90.000,C 0.000} C_DIS
LIN {X 275.544,Y 90.419,Z 155.797,A -161.833,B 90.000,C 0.000} C_DIS
LIN {X 275.490,Y 90.582,Z 155.919,A -161.799,B 90.000,C 0.000} C_DIS
LIN {X 275.259,Y 91.284,Z 156.767,A -161.653,B 90.000,C 0.000} C_DIS
LIN {X 275.205,Y 91.446,Z 156.872,A -161.619,B 90.000,C 0.000} C_DIS
LIN {X 275.034,Y 91.959,Z 157.423,A -161.512,B 90.000,C 0.000} C_DIS
LIN {X 275.007,Y 92.039,Z 157.563,A -161.496,B 90.000,C 0.000} C_DIS
LIN {X 275.751,Y 89.784,Z 156.780,A -161.965,B 90.000,C 0.000} C_DIS
LIN {X 276.227,Y 88.308,Z 156.127,A -162.271,B 90.000,C 0.000} C_DIS
LIN {X 276.245,Y 88.254,Z 156.112,A -162.282,B 90.000,C 0.000} C_DIS
LIN {X 276.911,Y 86.141,Z 154.955,A -162.720,B 90.000,C 0.000} C_DIS
LIN {X 277.122,Y 85.459,Z 154.490,A -162.861,B 90.000,C 0.000} C_DIS
LIN {X 277.214,Y 85.160,Z 154.314,A -162.923,B 90.000,C 0.000} C_DIS
LIN {X 277.658,Y 83.702,Z 153.239,A -163.224,B 90.000,C 0.000} C_DIS
LIN {X 277.694,Y 83.582,Z 153.097,A -163.249,B 90.000,C 0.000} C_DIS
LIN {X 277.760,Y 83.362,Z 152.926,A -163.294,B 90.000,C 0.000} C_DIS
LIN {X 278.289,Y 81.578,Z 151.257,A -163.662,B 90.000,C 0.000} C_DIS
LIN {X 278.395,Y 81.217,Z 150.847,A -163.736,B 90.000,C 0.000} C_DIS
LIN {X 278.450,Y 81.029,Z 150.681,A -163.775,B 90.000,C 0.000} C_DIS
LIN {X 278.858,Y 79.612,Z 148.943,A -164.066,B 90.000,C 0.000} C_DIS
LIN {X 278.867,Y 79.580,Z 148.836,A -164.073,B 90.000,C 0.000} C_DIS
LIN {X 278.876,Y 79.550,Z 148.801,A -164.079,B 90.000,C 0.000} C_DIS
LIN {X 278.894,Y 79.486,Z 148.742,A -164.092,B 90.000,C 0.000} C_DIS
LIN {X 278.961,Y 79.250,Z 148.383,A -164.141,B 90.000,C 0.000} C_DIS
LIN {X 278.969,Y 79.221,Z 148.346,A -164.147,B 90.000,C 0.000} C_DIS
LIN {X 278.988,Y 79.158,Z 148.281,A -164.160,B 90.000,C 0.000} C_DIS
LIN {X 279.057,Y 78.912,Z 147.948,A -164.210,B 90.000,C 0.000} C_DIS
LIN {X 279.228,Y 78.305,Z 147.023,A -164.335,B 90.000,C 0.000} C_DIS
LIN {X 279.433,Y 77.569,Z 145.696,A -164.486,B 90.000,C 0.000} C_DIS
LIN {X 279.497,Y 77.340,Z 145.331,A -164.533,B 90.000,C 0.000} C_DIS
LIN {X 279.507,Y 77.304,Z 145.217,A -164.540,B 90.000,C 0.000} C_DIS
LIN {X 279.570,Y 77.075,Z 144.851,A -164.587,B 90.000,C 0.000} C_DIS
LIN {X 279.608,Y 76.937,Z 144.591,A -164.615,B 90.000,C 0.000} C_DIS
LIN {X 279.645,Y 76.801,Z 144.237,A -164.643,B 90.000,C 0.000} C_DIS
LIN {X 279.661,Y 76.746,Z 144.136,A -164.654,B 90.000,C 0.000} C_DIS
LIN {X 279.674,Y 76.699,Z 144.093,A -164.664,B 90.000,C 0.000} C_DIS
LIN {X 279.725,Y 76.511,Z 143.681,A -164.702,B 90.000,C 0.000} C_DIS
LIN {X 279.728,Y 76.499,Z 143.624,A -164.705,B 90.000,C 0.000} C_DIS
LIN {X 279.783,Y 76.298,Z 143.169,A -164.746,B 90.000,C 0.000} C_DIS
LIN {X 279.793,Y 76.262,Z 143.055,A -164.754,B 90.000,C 0.000} C_DIS
LIN {X 279.858,Y 76.025,Z 142.576,A -164.802,B 90.000,C 0.000} C_DIS
LIN {X 279.870,Y 75.981,Z 142.372,A -164.811,B 90.000,C 0.000} C_DIS
LIN {X 279.914,Y 75.817,Z 142.087,A -164.845,B 90.000,C 0.000} C_DIS
LIN {X 279.926,Y 75.772,Z 141.860,A -164.854,B 90.000,C 0.000} C_DIS
LIN {X 280.105,Y 75.106,Z 140.147,A -164.990,B 90.000,C 0.000} C_DIS
LIN {X 280.196,Y 74.766,Z 139.072,A -165.060,B 90.000,C 0.000} C_DIS
LIN {X 280.200,Y 74.753,Z 138.958,A -165.062,B 90.000,C 0.000} C_DIS
LIN {X 280.250,Y 74.564,Z 138.335,A -165.101,B 90.000,C 0.000} C_DIS
LIN {X 280.399,Y 74.000,Z 135.904,A -165.216,B 90.000,C 0.000} C_DIS
LIN {X 280.451,Y 73.807,Z 135.089,A -165.256,B 90.000,C 0.000} C_DIS
LIN {X 280.459,Y 73.776,Z 135.032,A -165.262,B 90.000,C 0.000} C_DIS
LIN {X 280.468,Y 73.740,Z 134.919,A -165.269,B 90.000,C 0.000} C_DIS
LIN {X 280.486,Y 73.672,Z 134.520,A -165.283,B 90.000,C 0.000} C_DIS
LIN {X 280.495,Y 73.638,Z 134.470,A -165.290,B 90.000,C 0.000} C_DIS
LIN {X 280.537,Y 73.478,Z 133.266,A -165.323,B 90.000,C 0.000} C_DIS
LIN {X 280.544,Y 73.451,Z 133.212,A -165.328,B 90.000,C 0.000} C_DIS
LIN {X 280.588,Y 73.282,Z 132.074,A -165.363,B 90.000,C 0.000} C_DIS
LIN {X 280.608,Y 73.208,Z 131.377,A -165.378,B 90.000,C 0.000} C_DIS
LIN {X 280.617,Y 73.170,Z 131.220,A -165.386,B 90.000,C 0.000} C_DIS
LIN {X 280.636,Y 73.100,Z 130.438,A -165.400,B 90.000,C 0.000} C_DIS
LIN {X 280.654,Y 73.029,Z 130.097,A -165.415,B 90.000,C 0.000} C_DIS
LIN {X 280.700,Y 72.853,Z 127.603,A -165.451,B 90.000,C 0.000} C_DIS
LIN {X 280.715,Y 72.795,Z 125.104,A -165.462,B 90.000,C 0.000} C_DIS
LIN {X 280.712,Y 72.806,Z 123.555,A -165.460,B 90.000,C 0.000} C_DIS
LIN {X 280.723,Y 72.764,Z 123.364,A -165.469,B 90.000,C 0.000} C_DIS
LIN {X 280.696,Y 72.868,Z 122.008,A -165.447,B 90.000,C 0.000} C_DIS
LIN {X 280.702,Y 72.843,Z 121.946,A -165.452,B 90.000,C 0.000} C_DIS
LIN {X 280.710,Y 72.813,Z 121.894,A -165.459,B 90.000,C 0.000} C_DIS
LIN {X 280.653,Y 73.033,Z 119.452,A -165.414,B 90.000,C 0.000} C_DIS
LIN {X 278.717,Y 72.530,Z 119.452,A -165.414,B 90.000,C 0.000} C_DIS
WAIT SEC 0.1
RET=EKI_SetBool("oxy","torchState",FALSE)
RET = EKI_Send("oxy","torchState")
LIN {X 261.298,Y 67.997,Z 119.452,A -165.414,B 90.000,C 0.000} C_DIS
LIN {X 261.703,Y 66.418,Z 142.870,A -165.760,B 90.000,C 0.000} C_DIS
LIN {X 279.150,Y 70.846,Z 142.870,A -165.760,B 90.000,C 0.000} C_DIS
LIN {X 281.089,Y 71.338,Z 142.870,A -165.760,B 90.000,C 0.000} C_DIS
WAIT SEC 1
RET=EKI_SetBool("oxy","torchState",TRUE)
RET = EKI_Send("oxy","torchState")
LIN {X 281.105,Y 71.272,Z 144.079,A -165.773,B 90.000,C 0.000} C_DIS
LIN {X 281.098,Y 71.300,Z 144.136,A -165.767,B 90.000,C 0.000} C_DIS
LIN {X 281.093,Y 71.321,Z 144.203,A -165.763,B 90.000,C 0.000} C_DIS
LIN {X 281.095,Y 71.312,Z 146.703,A -165.765,B 90.000,C 0.000} C_DIS
LIN {X 281.090,Y 71.333,Z 149.203,A -165.761,B 90.000,C 0.000} C_DIS
LIN {X 281.074,Y 71.398,Z 151.702,A -165.747,B 90.000,C 0.000} C_DIS
LIN {X 281.048,Y 71.500,Z 154.200,A -165.727,B 90.000,C 0.000} C_DIS
LIN {X 281.015,Y 71.626,Z 156.696,A -165.701,B 90.000,C 0.000} C_DIS
LIN {X 280.973,Y 71.793,Z 159.190,A -165.667,B 90.000,C 0.000} C_DIS
LIN {X 280.969,Y 71.809,Z 159.427,A -165.663,B 90.000,C 0.000} C_DIS
LIN {X 280.907,Y 72.049,Z 161.914,A -165.615,B 90.000,C 0.000} C_DIS
LIN {X 280.899,Y 72.081,Z 162.328,A -165.608,B 90.000,C 0.000} C_DIS
LIN {X 280.839,Y 72.315,Z 164.490,A -165.560,B 90.000,C 0.000} C_DIS
LIN {X 280.827,Y 72.362,Z 164.675,A -165.551,B 90.000,C 0.000} C_DIS
LIN {X 280.765,Y 72.603,Z 166.780,A -165.502,B 90.000,C 0.000} C_DIS
LIN {X 280.750,Y 72.658,Z 166.908,A -165.490,B 90.000,C 0.000} C_DIS
LIN {X 280.711,Y 72.810,Z 168.331,A -165.459,B 90.000,C 0.000} C_DIS
LIN {X 280.692,Y 72.883,Z 168.560,A -165.444,B 90.000,C 0.000} C_DIS
LIN {X 280.667,Y 72.980,Z 169.513,A -165.425,B 90.000,C 0.000} C_DIS
LIN {X 280.659,Y 73.010,Z 169.598,A -165.418,B 90.000,C 0.000} C_DIS
LIN {X 280.640,Y 73.083,Z 169.939,A -165.403,B 90.000,C 0.000} C_DIS
LIN {X 280.542,Y 73.458,Z 172.409,A -165.327,B 90.000,C 0.000} C_DIS
LIN {X 280.494,Y 73.642,Z 173.606,A -165.289,B 90.000,C 0.000} C_DIS
LIN {X 280.487,Y 73.669,Z 173.665,A -165.284,B 90.000,C 0.000} C_DIS
LIN {X 280.473,Y 73.723,Z 173.920,A -165.273,B 90.000,C 0.000} C_DIS
LIN {X 280.465,Y 73.752,Z 174.005,A -165.267,B 90.000,C 0.000} C_DIS
LIN {X 280.393,Y 74.025,Z 175.602,A -165.211,B 90.000,C 0.000} C_DIS
LIN {X 280.387,Y 74.048,Z 175.656,A -165.206,B 90.000,C 0.000} C_DIS
LIN {X 280.261,Y 74.522,Z 178.102,A -165.110,B 90.000,C 0.000} C_DIS
LIN {X 280.253,Y 74.552,Z 178.160,A -165.103,B 90.000,C 0.000} C_DIS
LIN {X 280.216,Y 74.694,Z 178.900,A -165.074,B 90.000,C 0.000} C_DIS
LIN {X 280.065,Y 75.257,Z 181.330,A -164.959,B 90.000,C 0.000} C_DIS
LIN {X 279.974,Y 75.593,Z 182.662,A -164.890,B 90.000,C 0.000} C_DIS
LIN {X 279.925,Y 75.777,Z 183.115,A -164.853,B 90.000,C 0.000} C_DIS
LIN {X 279.293,Y 78.068,Z 183.892,A -164.383,B 90.000,C 0.000} C_DIS
LIN {X 278.894,Y 79.487,Z 184.275,A -164.092,B 90.000,C 0.000} C_DIS
LIN {X 278.858,Y 79.614,Z 184.328,A -164.066,B 90.000,C 0.000} C_DIS
LIN {X 278.173,Y 81.975,Z 184.787,A -163.580,B 90.000,C 0.000} C_DIS
LIN {X 277.462,Y 84.351,Z 185.099,A -163.090,B 90.000,C 0.000} C_DIS
LIN {X 276.722,Y 86.738,Z 185.154,A -162.596,B 90.000,C 0.000} C_DIS
LIN {X 275.966,Y 89.120,Z 185.081,A -162.103,B 90.000,C 0.000} C_DIS
LIN {X 275.725,Y 89.865,Z 185.032,A -161.948,B 90.000,C 0.000} C_DIS
LIN {X 275.155,Y 91.594,Z 184.786,A -161.588,B 90.000,C 0.000} C_DIS
LIN {X 275.133,Y 91.662,Z 184.751,A -161.574,B 90.000,C 0.000} C_DIS
LIN {X 275.035,Y 91.957,Z 184.666,A -161.513,B 90.000,C 0.000} C_DIS
LIN {X 274.677,Y 93.020,Z 184.467,A -161.291,B 90.000,C 0.000} C_DIS
LIN {X 274.109,Y 94.679,Z 183.835,A -160.945,B 90.000,C 0.000} C_DIS
LIN {X 274.072,Y 94.786,Z 183.809,A -160.922,B 90.000,C 0.000} C_DIS
LIN {X 274.035,Y 94.894,Z 183.796,A -160.900,B 90.000,C 0.000} C_DIS
LIN {X 273.853,Y 95.418,Z 183.548,A -160.790,B 90.000,C 0.000} C_DIS
LIN {X 273.829,Y 95.485,Z 183.533,A -160.776,B 90.000,C 0.000} C_DIS
LIN {X 273.717,Y 95.807,Z 183.340,A -160.709,B 90.000,C 0.000} C_DIS
LIN {X 273.642,Y 96.022,Z 183.286,A -160.664,B 90.000,C 0.000} C_DIS
LIN {X 273.320,Y 96.934,Z 182.815,A -160.473,B 90.000,C 0.000} C_DIS
LIN {X 273.163,Y 97.377,Z 182.645,A -160.380,B 90.000,C 0.000} C_DIS
LIN {X 273.148,Y 97.417,Z 182.588,A -160.371,B 90.000,C 0.000} C_DIS
LIN {X 273.137,Y 97.450,Z 182.556,A -160.365,B 90.000,C 0.000} C_DIS
LIN {X 272.976,Y 97.899,Z 182.345,A -160.270,B 90.000,C 0.000} C_DIS
LIN {X 272.860,Y 98.220,Z 182.146,A -160.203,B 90.000,C 0.000} C_DIS
LIN {X 272.783,Y 98.434,Z 182.083,A -160.158,B 90.000,C 0.000} C_DIS
LIN {X 272.662,Y 98.769,Z 181.858,A -160.088,B 90.000,C 0.000} C_DIS
LIN {X 272.414,Y 99.451,Z 181.494,A -159.944,B 90.000,C 0.000} C_DIS
LIN {X 272.325,Y 99.695,Z 181.346,A -159.893,B 90.000,C 0.000} C_DIS
LIN {X 272.285,Y 99.805,Z 181.249,A -159.870,B 90.000,C 0.000} C_DIS
LIN {X 272.216,Y 99.991,Z 181.200,A -159.831,B 90.000,C 0.000} C_DIS
LIN {X 272.150,Y 100.173,Z 181.119,A -159.792,B 90.000,C 0.000} C_DIS
LIN {X 272.109,Y 100.284,Z 181.035,A -159.769,B 90.000,C 0.000} C_DIS
LIN {X 272.050,Y 100.442,Z 180.948,A -159.736,B 90.000,C 0.000} C_DIS
LIN {X 272.022,Y 100.519,Z 180.887,A -159.720,B 90.000,C 0.000} C_DIS
LIN {X 271.983,Y 100.625,Z 180.837,A -159.697,B 90.000,C 0.000} C_DIS
LIN {X 271.923,Y 100.785,Z 180.717,A -159.663,B 90.000,C 0.000} C_DIS
LIN {X 271.884,Y 100.892,Z 180.666,A -159.641,B 90.000,C 0.000} C_DIS
LIN {X 271.857,Y 100.964,Z 180.606,A -159.626,B 90.000,C 0.000} C_DIS
LIN {X 271.712,Y 101.354,Z 180.379,A -159.544,B 90.000,C 0.000} C_DIS
LIN {X 271.685,Y 101.425,Z 180.318,A -159.528,B 90.000,C 0.000} C_DIS
LIN {X 271.645,Y 101.532,Z 180.268,A -159.506,B 90.000,C 0.000} C_DIS
LIN {X 271.619,Y 101.604,Z 180.208,A -159.491,B 90.000,C 0.000} C_DIS
LIN {X 271.160,Y 102.821,Z 179.358,A -159.234,B 90.000,C 0.000} C_DIS
LIN {X 271.043,Y 103.129,Z 179.175,A -159.169,B 90.000,C 0.000} C_DIS
LIN {X 271.023,Y 103.182,Z 179.127,A -159.157,B 90.000,C 0.000} C_DIS
LIN {X 270.423,Y 104.744,Z 177.973,A -158.827,B 90.000,C 0.000} C_DIS
LIN {X 270.389,Y 104.832,Z 177.875,A -158.808,B 90.000,C 0.000} C_DIS
LIN {X 270.338,Y 104.963,Z 177.804,A -158.780,B 90.000,C 0.000} C_DIS
LIN {X 269.686,Y 106.627,Z 176.325,A -158.427,B 90.000,C 0.000} C_DIS
LIN {X 269.603,Y 106.838,Z 176.168,A -158.383,B 90.000,C 0.000} C_DIS
LIN {X 269.562,Y 106.941,Z 175.998,A -158.361,B 90.000,C 0.000} C_DIS
LIN {X 269.136,Y 108.008,Z 174.973,A -158.134,B 90.000,C 0.000} C_DIS
LIN {X 269.116,Y 108.057,Z 174.888,A -158.123,B 90.000,C 0.000} C_DIS
LIN {X 269.053,Y 108.215,Z 174.716,A -158.090,B 90.000,C 0.000} C_DIS
LIN {X 268.989,Y 108.374,Z 174.484,A -158.056,B 90.000,C 0.000} C_DIS
LIN {X 268.957,Y 108.453,Z 174.405,A -158.039,B 90.000,C 0.000} C_DIS
LIN {X 268.925,Y 108.532,Z 174.346,A -158.022,B 90.000,C 0.000} C_DIS
LIN {X 268.562,Y 109.428,Z 173.138,A -157.831,B 90.000,C 0.000} C_DIS
LIN {X 268.107,Y 110.537,Z 171.332,A -157.594,B 90.000,C 0.000} C_DIS
LIN {X 267.733,Y 111.440,Z 169.031,A -157.401,B 90.000,C 0.000} C_DIS
LIN {X 267.682,Y 111.564,Z 168.630,A -157.375,B 90.000,C 0.000} C_DIS
LIN {X 267.674,Y 111.582,Z 168.501,A -157.371,B 90.000,C 0.000} C_DIS
LIN {X 267.699,Y 111.523,Z 168.529,A -157.383,B 90.000,C 0.000} C_DIS
LIN {X 267.746,Y 111.410,Z 168.563,A -157.408,B 90.000,C 0.000} C_DIS
LIN {X 268.003,Y 110.789,Z 169.056,A -157.540,B 90.000,C 0.000} C_DIS
LIN {X 268.052,Y 110.670,Z 169.127,A -157.566,B 90.000,C 0.000} C_DIS
LIN {X 268.791,Y 108.863,Z 170.689,A -157.952,B 90.000,C 0.000} C_DIS
LIN {X 268.990,Y 108.372,Z 171.105,A -158.056,B 90.000,C 0.000} C_DIS
LIN {X 269.010,Y 108.321,Z 171.171,A -158.067,B 90.000,C 0.000} C_DIS
LIN {X 269.023,Y 108.289,Z 171.203,A -158.074,B 90.000,C 0.000} C_DIS
LIN {X 269.368,Y 107.427,Z 171.901,A -158.257,B 90.000,C 0.000} C_DIS
LIN {X 269.404,Y 107.338,Z 171.999,A -158.276,B 90.000,C 0.000} C_DIS
LIN {X 269.536,Y 107.007,Z 172.242,A -158.347,B 90.000,C 0.000} C_DIS
LIN {X 269.559,Y 106.947,Z 172.303,A -158.359,B 90.000,C 0.000} C_DIS
LIN {X 269.579,Y 106.898,Z 172.330,A -158.370,B 90.000,C 0.000} C_DIS
LIN {X 269.645,Y 106.732,Z 172.496,A -158.405,B 90.000,C 0.000} C_DIS
LIN {X 269.664,Y 106.683,Z 172.513,A -158.416,B 90.000,C 0.000} C_DIS
LIN {X 270.143,Y 105.465,Z 173.498,A -158.674,B 90.000,C 0.000} C_DIS
LIN {X 270.174,Y 105.385,Z 173.551,A -158.691,B 90.000,C 0.000} C_DIS
LIN {X 270.205,Y 105.306,Z 173.617,A -158.708,B 90.000,C 0.000} C_DIS
LIN {X 270.217,Y 105.276,Z 173.652,A -158.714,B 90.000,C 0.000} C_DIS
LIN {X 270.657,Y 104.139,Z 174.461,A -158.955,B 90.000,C 0.000} C_DIS
LIN {X 270.677,Y 104.086,Z 174.517,A -158.966,B 90.000,C 0.000} C_DIS
LIN {X 270.792,Y 103.788,Z 174.730,A -159.029,B 90.000,C 0.000} C_DIS
LIN {X 270.922,Y 103.448,Z 174.909,A -159.101,B 90.000,C 0.000} C_DIS
LIN {X 270.967,Y 103.328,Z 175.006,A -159.127,B 90.000,C 0.000} C_DIS
LIN {X 271.023,Y 103.182,Z 175.084,A -159.157,B 90.000,C 0.000} C_DIS
LIN {X 271.109,Y 102.956,Z 175.251,A -159.205,B 90.000,C 0.000} C_DIS
LIN {X 271.185,Y 102.757,Z 175.443,A -159.247,B 90.000,C 0.000} C_DIS
LIN {X 271.325,Y 102.384,Z 175.668,A -159.326,B 90.000,C 0.000} C_DIS
LIN {X 271.344,Y 102.334,Z 175.713,A -159.337,B 90.000,C 0.000} C_DIS
LIN {X 271.491,Y 101.945,Z 175.836,A -159.419,B 90.000,C 0.000} C_DIS
LIN {X 271.506,Y 101.905,Z 175.878,A -159.427,B 90.000,C 0.000} C_DIS
LIN {X 271.631,Y 101.572,Z 176.112,A -159.498,B 90.000,C 0.000} C_DIS
LIN {X 271.892,Y 100.870,Z 176.467,A -159.645,B 90.000,C 0.000} C_DIS
LIN {X 271.904,Y 100.839,Z 176.500,A -159.652,B 90.000,C 0.000} C_DIS
LIN {X 271.922,Y 100.789,Z 176.567,A -159.663,B 90.000,C 0.000} C_DIS
LIN {X 272.066,Y 100.399,Z 176.690,A -159.745,B 90.000,C 0.000} C_DIS
LIN {X 272.081,Y 100.359,Z 176.737,A -159.753,B 90.000,C 0.000} C_DIS
LIN {X 272.109,Y 100.282,Z 176.794,A -159.769,B 90.000,C 0.000} C_DIS
LIN {X 272.199,Y 100.038,Z 176.933,A -159.821,B 90.000,C 0.000} C_DIS
LIN {X 272.224,Y 99.971,Z 176.948,A -159.835,B 90.000,C 0.000} C_DIS
LIN {X 272.414,Y 99.451,Z 177.198,A -159.944,B 90.000,C 0.000} C_DIS
LIN {X 272.492,Y 99.237,Z 177.246,A -159.989,B 90.000,C 0.000} C_DIS
LIN {X 272.725,Y 98.595,Z 177.551,A -160.124,B 90.000,C 0.000} C_DIS
LIN {X 272.803,Y 98.381,Z 177.590,A -160.169,B 90.000,C 0.000} C_DIS
LIN {X 273.100,Y 97.551,Z 177.896,A -160.343,B 90.000,C 0.000} C_DIS
LIN {X 273.172,Y 97.350,Z 177.940,A -160.386,B 90.000,C 0.000} C_DIS
LIN {X 273.310,Y 96.961,Z 178.066,A -160.467,B 90.000,C 0.000} C_DIS
LIN {X 273.453,Y 96.559,Z 178.200,A -160.551,B 90.000,C 0.000} C_DIS
LIN {X 273.547,Y 96.291,Z 178.233,A -160.608,B 90.000,C 0.000} C_DIS
LIN {X 273.585,Y 96.183,Z 178.270,A -160.630,B 90.000,C 0.000} C_DIS
LIN {X 273.603,Y 96.133,Z 178.304,A -160.641,B 90.000,C 0.000} C_DIS
LIN {X 273.914,Y 95.241,Z 178.423,A -160.827,B 90.000,C 0.000} C_DIS
LIN {X 273.942,Y 95.163,Z 178.447,A -160.844,B 90.000,C 0.000} C_DIS
LIN {X 274.751,Y 92.800,Z 178.552,A -161.337,B 90.000,C 0.000} C_DIS
LIN {X 274.934,Y 92.257,Z 178.542,A -161.450,B 90.000,C 0.000} C_DIS
LIN {X 275.618,Y 90.192,Z 178.163,A -161.880,B 90.000,C 0.000} C_DIS
LIN {X 276.335,Y 87.973,Z 177.262,A -162.341,B 90.000,C 0.000} C_DIS
LIN {X 276.374,Y 87.850,Z 177.188,A -162.366,B 90.000,C 0.000} C_DIS
LIN {X 276.385,Y 87.814,Z 177.135,A -162.374,B 90.000,C 0.000} C_DIS
LIN {X 276.708,Y 86.790,Z 176.562,A -162.586,B 90.000,C 0.000} C_DIS
LIN {X 276.742,Y 86.681,Z 176.513,A -162.608,B 90.000,C 0.000} C_DIS
LIN {X 277.002,Y 85.847,Z 175.884,A -162.781,B 90.000,C 0.000} C_DIS
LIN {X 277.118,Y 85.474,Z 175.656,A -162.858,B 90.000,C 0.000} C_DIS
LIN {X 277.126,Y 85.446,Z 175.542,A -162.864,B 90.000,C 0.000} C_DIS
LIN {X 277.567,Y 84.005,Z 174.291,A -163.162,B 90.000,C 0.000} C_DIS
LIN {X 277.577,Y 83.969,Z 174.177,A -163.169,B 90.000,C 0.000} C_DIS
LIN {X 278.065,Y 82.341,Z 172.343,A -163.505,B 90.000,C 0.000} C_DIS
LIN {X 278.179,Y 81.955,Z 171.866,A -163.584,B 90.000,C 0.000} C_DIS
LIN {X 278.358,Y 81.344,Z 170.993,A -163.710,B 90.000,C 0.000} C_DIS
LIN {X 278.386,Y 81.249,Z 170.901,A -163.730,B 90.000,C 0.000} C_DIS
LIN {X 278.425,Y 81.116,Z 170.615,A -163.757,B 90.000,C 0.000} C_DIS
LIN {X 278.537,Y 80.727,Z 170.097,A -163.837,B 90.000,C 0.000} C_DIS
LIN {X 278.573,Y 80.604,Z 169.809,A -163.862,B 90.000,C 0.000} C_DIS
LIN {X 278.788,Y 79.856,Z 168.667,A -164.016,B 90.000,C 0.000} C_DIS
LIN {X 278.863,Y 79.595,Z 168.166,A -164.070,B 90.000,C 0.000} C_DIS
LIN {X 278.928,Y 79.367,Z 167.805,A -164.117,B 90.000,C 0.000} C_DIS
LIN {X 278.933,Y 79.349,Z 167.748,A -164.120,B 90.000,C 0.000} C_DIS
LIN {X 278.936,Y 79.339,Z 167.691,A -164.123,B 90.000,C 0.000} C_DIS
LIN {X 279.039,Y 78.976,Z 167.008,A -164.197,B 90.000,C 0.000} C_DIS
LIN {X 279.042,Y 78.966,Z 166.951,A -164.199,B 90.000,C 0.000} C_DIS
LIN {X 279.049,Y 78.942,Z 166.894,A -164.204,B 90.000,C 0.000} C_DIS
LIN {X 279.065,Y 78.884,Z 166.813,A -164.216,B 90.000,C 0.000} C_DIS
LIN {X 279.105,Y 78.741,Z 166.553,A -164.245,B 90.000,C 0.000} C_DIS
LIN {X 279.204,Y 78.391,Z 165.827,A -164.317,B 90.000,C 0.000} C_DIS
LIN {X 279.218,Y 78.342,Z 165.756,A -164.327,B 90.000,C 0.000} C_DIS
LIN {X 279.407,Y 77.664,Z 164.277,A -164.466,B 90.000,C 0.000} C_DIS
LIN {X 279.411,Y 77.651,Z 164.220,A -164.469,B 90.000,C 0.000} C_DIS
LIN {X 279.466,Y 77.450,Z 163.765,A -164.510,B 90.000,C 0.000} C_DIS
LIN {X 279.476,Y 77.416,Z 163.651,A -164.517,B 90.000,C 0.000} C_DIS
LIN {X 279.541,Y 77.179,Z 163.196,A -164.566,B 90.000,C 0.000} C_DIS
LIN {X 279.556,Y 77.127,Z 162.968,A -164.576,B 90.000,C 0.000} C_DIS
LIN {X 279.570,Y 77.075,Z 162.887,A -164.587,B 90.000,C 0.000} C_DIS
LIN {X 279.608,Y 76.939,Z 162.570,A -164.615,B 90.000,C 0.000} C_DIS
LIN {X 279.617,Y 76.906,Z 162.456,A -164.622,B 90.000,C 0.000} C_DIS
LIN {X 279.637,Y 76.832,Z 162.300,A -164.637,B 90.000,C 0.000} C_DIS
LIN {X 279.626,Y 76.872,Z 162.173,A -164.628,B 90.000,C 0.000} C_DIS
LIN {X 279.319,Y 77.981,Z 163.082,A -164.401,B 90.000,C 0.000} C_DIS
LIN {X 279.304,Y 78.035,Z 163.139,A -164.390,B 90.000,C 0.000} C_DIS
LIN {X 279.300,Y 78.048,Z 163.196,A -164.387,B 90.000,C 0.000} C_DIS
LIN {X 279.146,Y 78.596,Z 163.594,A -164.275,B 90.000,C 0.000} C_DIS
LIN {X 279.071,Y 78.863,Z 163.790,A -164.220,B 90.000,C 0.000} C_DIS
LIN {X 279.042,Y 78.965,Z 163.880,A -164.199,B 90.000,C 0.000} C_DIS
LIN {X 279.036,Y 78.986,Z 163.936,A -164.195,B 90.000,C 0.000} C_DIS
LIN {X 279.000,Y 79.114,Z 164.007,A -164.169,B 90.000,C 0.000} C_DIS
LIN {X 278.604,Y 80.497,Z 165.018,A -163.884,B 90.000,C 0.000} C_DIS
LIN {X 278.517,Y 80.798,Z 165.193,A -163.822,B 90.000,C 0.000} C_DIS
LIN {X 277.915,Y 82.846,Z 166.495,A -163.401,B 90.000,C 0.000} C_DIS
LIN {X 277.273,Y 84.969,Z 167.649,A -162.963,B 90.000,C 0.000} C_DIS
LIN {X 276.589,Y 87.170,Z 168.616,A -162.507,B 90.000,C 0.000} C_DIS
LIN {X 275.861,Y 89.446,Z 169.351,A -162.035,B 90.000,C 0.000} C_DIS
LIN {X 275.099,Y 91.762,Z 169.900,A -161.553,B 90.000,C 0.000} C_DIS
LIN {X 274.336,Y 94.020,Z 170.161,A -161.082,B 90.000,C 0.000} C_DIS
LIN {X 273.515,Y 96.378,Z 170.039,A -160.589,B 90.000,C 0.000} C_DIS
LIN {X 273.152,Y 97.406,Z 169.947,A -160.374,B 90.000,C 0.000} C_DIS
LIN {X 273.110,Y 97.524,Z 169.913,A -160.349,B 90.000,C 0.000} C_DIS
LIN {X 273.091,Y 97.577,Z 169.881,A -160.338,B 90.000,C 0.000} C_DIS
LIN {X 272.340,Y 99.654,Z 169.342,A -159.902,B 90.000,C 0.000} C_DIS
LIN {X 272.296,Y 99.774,Z 169.325,A -159.876,B 90.000,C 0.000} C_DIS
LIN {X 272.236,Y 99.937,Z 169.259,A -159.842,B 90.000,C 0.000} C_DIS
LIN {X 272.202,Y 100.031,Z 169.246,A -159.822,B 90.000,C 0.000} C_DIS
LIN {X 271.705,Y 101.372,Z 168.651,A -159.540,B 90.000,C 0.000} C_DIS
LIN {X 271.690,Y 101.412,Z 168.610,A -159.531,B 90.000,C 0.000} C_DIS
LIN {X 271.504,Y 101.909,Z 168.419,A -159.426,B 90.000,C 0.000} C_DIS
LIN {X 271.394,Y 102.202,Z 168.260,A -159.365,B 90.000,C 0.000} C_DIS
LIN {X 271.366,Y 102.278,Z 168.199,A -159.349,B 90.000,C 0.000} C_DIS
LIN {X 271.325,Y 102.384,Z 168.149,A -159.326,B 90.000,C 0.000} C_DIS
LIN {X 271.297,Y 102.460,Z 168.089,A -159.310,B 90.000,C 0.000} C_DIS
LIN {X 271.168,Y 102.799,Z 167.894,A -159.238,B 90.000,C 0.000} C_DIS
LIN {X 271.124,Y 102.916,Z 167.797,A -159.214,B 90.000,C 0.000} C_DIS
LIN {X 270.995,Y 103.256,Z 167.618,A -159.142,B 90.000,C 0.000} C_DIS
LIN {X 270.854,Y 103.626,Z 167.349,A -159.064,B 90.000,C 0.000} C_DIS
LIN {X 270.649,Y 104.160,Z 166.980,A -158.951,B 90.000,C 0.000} C_DIS
LIN {X 270.588,Y 104.317,Z 166.876,A -158.917,B 90.000,C 0.000} C_DIS
LIN {X 270.500,Y 104.545,Z 166.685,A -158.869,B 90.000,C 0.000} C_DIS
LIN {X 270.440,Y 104.702,Z 166.580,A -158.836,B 90.000,C 0.000} C_DIS
LIN {X 270.380,Y 104.856,Z 166.439,A -158.803,B 90.000,C 0.000} C_DIS
LIN {X 270.338,Y 104.963,Z 166.368,A -158.780,B 90.000,C 0.000} C_DIS
LIN {X 269.651,Y 106.716,Z 164.724,A -158.408,B 90.000,C 0.000} C_DIS
LIN {X 269.328,Y 107.529,Z 163.824,A -158.236,B 90.000,C 0.000} C_DIS
LIN {X 269.307,Y 107.582,Z 163.793,A -158.224,B 90.000,C 0.000} C_DIS
LIN {X 269.286,Y 107.635,Z 163.771,A -158.213,B 90.000,C 0.000} C_DIS
LIN {X 269.138,Y 108.004,Z 163.258,A -158.135,B 90.000,C 0.000} C_DIS
LIN {X 269.116,Y 108.057,Z 163.224,A -158.123,B 90.000,C 0.000} C_DIS
LIN {X 269.095,Y 108.110,Z 163.207,A -158.112,B 90.000,C 0.000} C_DIS
LIN {X 268.898,Y 108.599,Z 162.570,A -158.008,B 90.000,C 0.000} C_DIS
LIN {X 268.785,Y 108.879,Z 162.072,A -157.948,B 90.000,C 0.000} C_DIS
LIN {X 268.797,Y 108.849,Z 162.104,A -157.955,B 90.000,C 0.000} C_DIS
LIN {X 268.903,Y 108.587,Z 162.213,A -158.010,B 90.000,C 0.000} C_DIS
LIN {X 268.951,Y 108.469,Z 162.228,A -158.036,B 90.000,C 0.000} C_DIS
LIN {X 269.842,Y 106.228,Z 162.886,A -158.512,B 90.000,C 0.000} C_DIS
LIN {X 270.431,Y 104.723,Z 163.274,A -158.831,B 90.000,C 0.000} C_DIS
LIN {X 270.646,Y 104.168,Z 163.388,A -158.949,B 90.000,C 0.000} C_DIS
LIN {X 270.982,Y 103.289,Z 163.509,A -159.135,B 90.000,C 0.000} C_DIS
LIN {X 271.043,Y 103.130,Z 163.567,A -159.168,B 90.000,C 0.000} C_DIS
LIN {X 271.916,Y 100.805,Z 163.850,A -159.659,B 90.000,C 0.000} C_DIS
LIN {X 272.773,Y 98.461,Z 163.991,A -160.152,B 90.000,C 0.000} C_DIS
LIN {X 273.298,Y 96.996,Z 163.969,A -160.460,B 90.000,C 0.000} C_DIS
LIN {X 273.320,Y 96.934,Z 163.993,A -160.473,B 90.000,C 0.000} C_DIS
LIN {X 273.361,Y 96.819,Z 164.018,A -160.497,B 90.000,C 0.000} C_DIS
LIN {X 273.809,Y 95.545,Z 163.911,A -160.764,B 90.000,C 0.000} C_DIS
LIN {X 273.829,Y 95.485,Z 163.928,A -160.776,B 90.000,C 0.000} C_DIS
LIN {X 274.639,Y 93.132,Z 163.684,A -161.268,B 90.000,C 0.000} C_DIS
LIN {X 275.416,Y 90.803,Z 163.215,A -161.753,B 90.000,C 0.000} C_DIS
LIN {X 276.162,Y 88.512,Z 162.548,A -162.229,B 90.000,C 0.000} C_DIS
LIN {X 276.867,Y 86.283,Z 161.664,A -162.691,B 90.000,C 0.000} C_DIS
LIN {X 277.464,Y 84.343,Z 160.687,A -163.092,B 90.000,C 0.000} C_DIS
LIN {X 277.518,Y 84.166,Z 160.549,A -163.128,B 90.000,C 0.000} C_DIS
LIN {X 277.852,Y 83.055,Z 159.896,A -163.358,B 90.000,C 0.000} C_DIS
LIN {X 277.963,Y 82.682,Z 159.611,A -163.435,B 90.000,C 0.000} C_DIS
LIN {X 278.053,Y 82.381,Z 159.408,A -163.497,B 90.000,C 0.000} C_DIS
LIN {X 278.074,Y 82.308,Z 159.327,A -163.512,B 90.000,C 0.000} C_DIS
LIN {X 278.130,Y 82.120,Z 159.228,A -163.550,B 90.000,C 0.000} C_DIS
LIN {X 278.541,Y 80.715,Z 158.078,A -163.840,B 90.000,C 0.000} C_DIS
LIN {X 278.850,Y 79.640,Z 157.165,A -164.061,B 90.000,C 0.000} C_DIS
LIN {X 278.857,Y 79.615,Z 157.120,A -164.066,B 90.000,C 0.000} C_DIS
LIN {X 278.960,Y 79.253,Z 156.708,A -164.140,B 90.000,C 0.000} C_DIS
LIN {X 279.162,Y 78.542,Z 156.027,A -164.286,B 90.000,C 0.000} C_DIS
LIN {X 279.577,Y 77.050,Z 154.146,A -164.592,B 90.000,C 0.000} C_DIS
LIN {X 279.601,Y 76.962,Z 154.063,A -164.610,B 90.000,C 0.000} C_DIS
LIN {X 279.625,Y 76.875,Z 153.997,A -164.628,B 90.000,C 0.000} C_DIS
LIN {X 279.926,Y 75.771,Z 152.329,A -164.854,B 90.000,C 0.000} C_DIS
LIN {X 280.023,Y 75.412,Z 151.874,A -164.927,B 90.000,C 0.000} C_DIS
LIN {X 280.026,Y 75.401,Z 151.817,A -164.930,B 90.000,C 0.000} C_DIS
LIN {X 280.031,Y 75.383,Z 151.760,A -164.933,B 90.000,C 0.000} C_DIS
LIN {X 280.093,Y 75.154,Z 151.399,A -164.980,B 90.000,C 0.000} C_DIS
LIN {X 280.152,Y 74.934,Z 150.983,A -165.025,B 90.000,C 0.000} C_DIS
LIN {X 280.167,Y 74.876,Z 150.907,A -165.037,B 90.000,C 0.000} C_DIS
LIN {X 280.180,Y 74.827,Z 150.793,A -165.047,B 90.000,C 0.000} C_DIS
LIN {X 280.211,Y 74.711,Z 150.622,A -165.071,B 90.000,C 0.000} C_DIS
LIN {X 280.224,Y 74.662,Z 150.508,A -165.081,B 90.000,C 0.000} C_DIS
LIN {X 280.240,Y 74.604,Z 150.427,A -165.093,B 90.000,C 0.000} C_DIS
LIN {X 280.530,Y 73.504,Z 148.201,A -165.318,B 90.000,C 0.000} C_DIS
LIN {X 280.605,Y 73.219,Z 147.607,A -165.376,B 90.000,C 0.000} C_DIS
LIN {X 280.662,Y 72.999,Z 147.095,A -165.421,B 90.000,C 0.000} C_DIS
LIN {X 280.671,Y 72.965,Z 146.981,A -165.427,B 90.000,C 0.000} C_DIS
LIN {X 280.733,Y 72.724,Z 146.435,A -165.477,B 90.000,C 0.000} C_DIS
LIN {X 280.736,Y 72.715,Z 146.335,A -165.479,B 90.000,C 0.000} C_DIS
LIN {X 280.767,Y 72.594,Z 146.113,A -165.503,B 90.000,C 0.000} C_DIS
LIN {X 280.809,Y 72.430,Z 145.629,A -165.537,B 90.000,C 0.000} C_DIS
LIN {X 280.890,Y 72.117,Z 144.842,A -165.601,B 90.000,C 0.000} C_DIS
LIN {X 280.892,Y 72.109,Z 144.742,A -165.602,B 90.000,C 0.000} C_DIS
LIN {X 280.973,Y 71.793,Z 143.908,A -165.667,B 90.000,C 0.000} C_DIS
LIN {X 280.985,Y 71.746,Z 143.681,A -165.676,B 90.000,C 0.000} C_DIS
LIN {X 281.050,Y 71.489,Z 142.927,A -165.729,B 90.000,C 0.000} C_DIS
LIN {X 281.070,Y 71.412,Z 142.776,A -165.744,B 90.000,C 0.000} C_DIS
LIN {X 281.089,Y 71.338,Z 142.870,A -165.760,B 90.000,C 0.000} C_DIS
LIN {X 279.150,Y 70.846,Z 142.870,A -165.760,B 90.000,C 0.000} C_DIS
WAIT SEC 0.1
RET=EKI_SetBool("oxy","torchState",FALSE)
RET = EKI_Send("oxy","torchState")
LIN {X 261.703,Y 66.418,Z 142.870,A -165.760,B 90.000,C 0.000} C_DIS
LIN {X 256.400,Y 84.611,Z 140.333,A -161.737,B 90.000,C 0.000} C_DIS
LIN {X 273.493,Y 90.252,Z 140.333,A -161.737,B 90.000,C 0.000} C_DIS
LIN {X 275.393,Y 90.879,Z 140.333,A -161.737,B 90.000,C 0.000} C_DIS
WAIT SEC 1
RET=EKI_SetBool("oxy","torchState",TRUE)
RET = EKI_Send("oxy","torchState")
LIN {X 275.264,Y 91.267,Z 142.159,A -161.656,B 90.000,C 0.000} C_DIS
LIN {X 275.238,Y 91.347,Z 142.315,A -161.640,B 90.000,C 0.000} C_DIS
LIN {X 275.226,Y 91.382,Z 142.429,A -161.632,B 90.000,C 0.000} C_DIS
LIN {X 275.151,Y 91.609,Z 142.970,A -161.585,B 90.000,C 0.000} C_DIS
LIN {X 275.143,Y 91.632,Z 143.059,A -161.580,B 90.000,C 0.000} C_DIS
LIN {X 275.136,Y 91.653,Z 143.112,A -161.576,B 90.000,C 0.000} C_DIS
LIN {X 275.080,Y 91.822,Z 143.396,A -161.541,B 90.000,C 0.000} C_DIS
LIN {X 275.062,Y 91.875,Z 143.624,A -161.530,B 90.000,C 0.000} C_DIS
LIN {X 274.989,Y 92.093,Z 143.985,A -161.484,B 90.000,C 0.000} C_DIS
LIN {X 274.916,Y 92.309,Z 144.401,A -161.439,B 90.000,C 0.000} C_DIS
LIN {X 274.767,Y 92.754,Z 145.046,A -161.347,B 90.000,C 0.000} C_DIS
LIN {X 274.753,Y 92.795,Z 145.132,A -161.338,B 90.000,C 0.000} C_DIS
LIN {X 274.734,Y 92.852,Z 145.217,A -161.326,B 90.000,C 0.000} C_DIS
LIN {X 274.725,Y 92.878,Z 145.270,A -161.321,B 90.000,C 0.000} C_DIS
LIN {X 274.672,Y 93.035,Z 145.449,A -161.288,B 90.000,C 0.000} C_DIS
LIN {X 274.663,Y 93.061,Z 145.502,A -161.283,B 90.000,C 0.000} C_DIS
LIN {X 274.644,Y 93.118,Z 145.562,A -161.271,B 90.000,C 0.000} C_DIS
LIN {X 274.442,Y 93.710,Z 146.365,A -161.147,B 90.000,C 0.000} C_DIS
LIN {X 274.387,Y 93.872,Z 146.470,A -161.113,B 90.000,C 0.000} C_DIS
LIN {X 274.236,Y 94.310,Z 146.924,A -161.022,B 90.000,C 0.000} C_DIS
LIN {X 274.224,Y 94.346,Z 147.038,A -161.014,B 90.000,C 0.000} C_DIS
LIN {X 274.051,Y 94.847,Z 147.436,A -160.910,B 90.000,C 0.000} C_DIS
LIN {X 274.043,Y 94.870,Z 147.489,A -160.905,B 90.000,C 0.000} C_DIS
LIN {X 274.017,Y 94.947,Z 147.578,A -160.889,B 90.000,C 0.000} C_DIS
LIN {X 273.941,Y 95.164,Z 147.749,A -160.843,B 90.000,C 0.000} C_DIS
LIN {X 273.914,Y 95.242,Z 147.837,A -160.827,B 90.000,C 0.000} C_DIS
LIN {X 273.877,Y 95.349,Z 147.924,A -160.805,B 90.000,C 0.000} C_DIS
LIN {X 273.829,Y 95.485,Z 148.013,A -160.776,B 90.000,C 0.000} C_DIS
LIN {X 273.798,Y 95.575,Z 148.102,A -160.757,B 90.000,C 0.000} C_DIS
LIN {X 273.599,Y 96.144,Z 148.517,A -160.638,B 90.000,C 0.000} C_DIS
LIN {X 273.593,Y 96.159,Z 148.569,A -160.635,B 90.000,C 0.000} C_DIS
LIN {X 273.491,Y 96.452,Z 148.751,A -160.574,B 90.000,C 0.000} C_DIS
LIN {X 273.370,Y 96.792,Z 149.029,A -160.502,B 90.000,C 0.000} C_DIS
LIN {X 273.245,Y 97.144,Z 149.257,A -160.429,B 90.000,C 0.000} C_DIS
LIN {X 273.220,Y 97.215,Z 149.897,A -160.414,B 90.000,C 0.000} C_DIS
LIN {X 273.244,Y 97.149,Z 150.537,A -160.428,B 90.000,C 0.000} C_DIS
LIN {X 273.355,Y 96.836,Z 151.058,A -160.493,B 90.000,C 0.000} C_DIS
LIN {X 273.496,Y 96.435,Z 151.313,A -160.577,B 90.000,C 0.000} C_DIS
LIN {X 273.686,Y 95.895,Z 151.376,A -160.690,B 90.000,C 0.000} C_DIS
LIN {X 274.072,Y 94.787,Z 151.345,A -160.922,B 90.000,C 0.000} C_DIS
LIN {X 273.792,Y 95.593,Z 152.553,A -160.754,B 90.000,C 0.000} C_DIS
LIN {X 273.772,Y 95.650,Z 152.614,A -160.742,B 90.000,C 0.000} C_DIS
LIN {X 273.763,Y 95.676,Z 152.667,A -160.736,B 90.000,C 0.000} C_DIS
LIN {X 273.736,Y 95.754,Z 152.756,A -160.720,B 90.000,C 0.000} C_DIS
LIN {X 273.705,Y 95.841,Z 152.831,A -160.702,B 90.000,C 0.000} C_DIS
LIN {X 273.687,Y 95.894,Z 152.943,A -160.691,B 90.000,C 0.000} C_DIS
LIN {X 273.660,Y 95.971,Z 152.972,A -160.675,B 90.000,C 0.000} C_DIS
LIN {X 273.586,Y 96.181,Z 153.240,A -160.631,B 90.000,C 0.000} C_DIS
LIN {X 273.299,Y 96.993,Z 154.008,A -160.460,B 90.000,C 0.000} C_DIS
LIN {X 273.246,Y 97.143,Z 154.093,A -160.429,B 90.000,C 0.000} C_DIS
LIN {X 273.234,Y 97.176,Z 154.150,A -160.422,B 90.000,C 0.000} C_DIS
LIN {X 273.229,Y 97.191,Z 154.207,A -160.419,B 90.000,C 0.000} C_DIS
LIN {X 273.097,Y 97.559,Z 154.434,A -160.342,B 90.000,C 0.000} C_DIS
LIN {X 273.046,Y 97.703,Z 154.605,A -160.311,B 90.000,C 0.000} C_DIS
LIN {X 272.905,Y 98.096,Z 154.833,A -160.229,B 90.000,C 0.000} C_DIS
LIN {X 272.144,Y 100.189,Z 155.970,A -159.789,B 90.000,C 0.000} C_DIS
LIN {X 271.309,Y 102.424,Z 156.717,A -159.318,B 90.000,C 0.000} C_DIS
LIN {X 270.430,Y 104.725,Z 157.139,A -158.831,B 90.000,C 0.000} C_DIS
LIN {X 270.267,Y 105.145,Z 157.159,A -158.742,B 90.000,C 0.000} C_DIS
LIN {X 270.299,Y 105.064,Z 157.026,A -158.759,B 90.000,C 0.000} C_DIS
LIN {X 270.370,Y 104.881,Z 156.429,A -158.798,B 90.000,C 0.000} C_DIS
LIN {X 270.402,Y 104.799,Z 155.874,A -158.815,B 90.000,C 0.000} C_DIS
LIN {X 270.413,Y 104.771,Z 155.800,A -158.821,B 90.000,C 0.000} C_DIS
LIN {X 270.423,Y 104.746,Z 155.749,A -158.827,B 90.000,C 0.000} C_DIS
LIN {X 270.402,Y 104.798,Z 155.293,A -158.815,B 90.000,C 0.000} C_DIS
LIN {X 270.340,Y 104.958,Z 154.579,A -158.782,B 90.000,C 0.000} C_DIS
LIN {X 270.287,Y 105.094,Z 154.219,A -158.753,B 90.000,C 0.000} C_DIS
LIN {X 270.205,Y 105.306,Z 153.828,A -158.708,B 90.000,C 0.000} C_DIS
LIN {X 270.143,Y 105.465,Z 153.665,A -158.674,B 90.000,C 0.000} C_DIS
LIN {X 270.059,Y 105.680,Z 153.353,A -158.629,B 90.000,C 0.000} C_DIS
LIN {X 269.935,Y 105.995,Z 153.091,A -158.562,B 90.000,C 0.000} C_DIS
LIN {X 269.706,Y 106.577,Z 152.715,A -158.438,B 90.000,C 0.000} C_DIS
LIN {X 269.664,Y 106.683,Z 152.687,A -158.416,B 90.000,C 0.000} C_DIS
LIN {X 269.622,Y 106.789,Z 152.672,A -158.393,B 90.000,C 0.000} C_DIS
LIN {X 269.527,Y 107.028,Z 152.564,A -158.342,B 90.000,C 0.000} C_DIS
LIN {X 269.271,Y 107.673,Z 152.481,A -158.205,B 90.000,C 0.000} C_DIS
LIN {X 268.811,Y 108.814,Z 152.710,A -157.962,B 90.000,C 0.000} C_DIS
LIN {X 268.680,Y 109.139,Z 152.865,A -157.893,B 90.000,C 0.000} C_DIS
LIN {X 268.386,Y 109.858,Z 153.441,A -157.739,B 90.000,C 0.000} C_DIS
LIN {X 268.351,Y 109.944,Z 153.501,A -157.721,B 90.000,C 0.000} C_DIS
LIN {X 268.336,Y 109.981,Z 153.581,A -157.713,B 90.000,C 0.000} C_DIS
LIN {X 268.239,Y 110.218,Z 153.915,A -157.662,B 90.000,C 0.000} C_DIS
LIN {X 268.216,Y 110.274,Z 153.979,A -157.650,B 90.000,C 0.000} C_DIS
LIN {X 268.206,Y 110.297,Z 154.036,A -157.646,B 90.000,C 0.000} C_DIS
LIN {X 268.200,Y 110.312,Z 154.093,A -157.642,B 90.000,C 0.000} C_DIS
LIN {X 268.091,Y 110.577,Z 154.704,A -157.586,B 90.000,C 0.000} C_DIS
LIN {X 268.039,Y 110.704,Z 155.691,A -157.559,B 90.000,C 0.000} C_DIS
LIN {X 268.139,Y 110.461,Z 157.039,A -157.611,B 90.000,C 0.000} C_DIS
LIN {X 268.135,Y 110.471,Z 157.124,A -157.608,B 90.000,C 0.000} C_DIS
LIN {X 268.113,Y 110.524,Z 157.078,A -157.597,B 90.000,C 0.000} C_DIS
LIN {X 268.033,Y 110.718,Z 157.016,A -157.556,B 90.000,C 0.000} C_DIS
LIN {X 267.276,Y 112.533,Z 156.741,A -157.167,B 90.000,C 0.000} C_DIS
LIN {X 267.255,Y 112.582,Z 156.717,A -157.157,B 90.000,C 0.000} C_DIS
LIN {X 267.207,Y 112.696,Z 156.684,A -157.132,B 90.000,C 0.000} C_DIS
LIN {X 266.653,Y 114.002,Z 156.458,A -156.852,B 90.000,C 0.000} C_DIS
LIN {X 266.633,Y 114.049,Z 156.423,A -156.842,B 90.000,C 0.000} C_DIS
LIN {X 266.588,Y 114.153,Z 156.385,A -156.819,B 90.000,C 0.000} C_DIS
LIN {X 266.543,Y 114.258,Z 156.373,A -156.797,B 90.000,C 0.000} C_DIS
LIN {X 266.273,Y 114.885,Z 156.087,A -156.662,B 90.000,C 0.000} C_DIS
LIN {X 266.183,Y 115.094,Z 156.037,A -156.617,B 90.000,C 0.000} C_DIS
LIN {X 266.041,Y 115.422,Z 155.869,A -156.546,B 90.000,C 0.000} C_DIS
LIN {X 265.988,Y 115.543,Z 155.774,A -156.520,B 90.000,C 0.000} C_DIS
LIN {X 265.921,Y 115.698,Z 155.686,A -156.487,B 90.000,C 0.000} C_DIS
LIN {X 265.889,Y 115.773,Z 155.629,A -156.471,B 90.000,C 0.000} C_DIS
LIN {X 265.872,Y 115.812,Z 155.582,A -156.462,B 90.000,C 0.000} C_DIS
LIN {X 265.337,Y 117.031,Z 154.719,A -156.199,B 90.000,C 0.000} C_DIS
LIN {X 265.294,Y 117.128,Z 154.548,A -156.179,B 90.000,C 0.000} C_DIS
LIN {X 265.041,Y 117.700,Z 153.913,A -156.055,B 90.000,C 0.000} C_DIS
LIN {X 265.018,Y 117.752,Z 153.894,A -156.044,B 90.000,C 0.000} C_DIS
LIN {X 264.995,Y 117.804,Z 153.840,A -156.032,B 90.000,C 0.000} C_DIS
LIN {X 264.870,Y 118.085,Z 153.392,A -155.972,B 90.000,C 0.000} C_DIS
LIN {X 264.555,Y 118.788,Z 151.874,A -155.819,B 90.000,C 0.000} C_DIS
LIN {X 264.379,Y 119.180,Z 150.213,A -155.734,B 90.000,C 0.000} C_DIS
LIN {X 264.350,Y 119.245,Z 147.714,A -155.721,B 90.000,C 0.000} C_DIS
LIN {X 264.382,Y 119.173,Z 146.692,A -155.736,B 90.000,C 0.000} C_DIS
LIN {X 264.438,Y 119.049,Z 146.302,A -155.763,B 90.000,C 0.000} C_DIS
LIN {X 264.725,Y 118.409,Z 145.199,A -155.901,B 90.000,C 0.000} C_DIS
LIN {X 264.762,Y 118.326,Z 145.133,A -155.919,B 90.000,C 0.000} C_DIS
LIN {X 264.834,Y 118.164,Z 144.960,A -155.954,B 90.000,C 0.000} C_DIS
LIN {X 264.871,Y 118.081,Z 144.894,A -155.972,B 90.000,C 0.000} C_DIS
LIN {X 264.965,Y 117.870,Z 144.648,A -156.018,B 90.000,C 0.000} C_DIS
LIN {X 264.995,Y 117.804,Z 144.601,A -156.032,B 90.000,C 0.000} C_DIS
LIN {X 265.444,Y 116.787,Z 143.513,A -156.252,B 90.000,C 0.000} C_DIS
LIN {X 265.845,Y 115.872,Z 142.685,A -156.449,B 90.000,C 0.000} C_DIS
LIN {X 265.908,Y 115.727,Z 142.600,A -156.481,B 90.000,C 0.000} C_DIS
LIN {X 266.076,Y 115.342,Z 142.259,A -156.564,B 90.000,C 0.000} C_DIS
LIN {X 266.391,Y 114.611,Z 141.690,A -156.721,B 90.000,C 0.000} C_DIS
LIN {X 266.999,Y 113.188,Z 140.603,A -157.027,B 90.000,C 0.000} C_DIS
LIN {X 267.018,Y 113.144,Z 140.552,A -157.036,B 90.000,C 0.000} C_DIS
LIN {X 267.181,Y 112.758,Z 140.324,A -157.119,B 90.000,C 0.000} C_DIS
LIN {X 267.989,Y 110.823,Z 138.963,A -157.533,B 90.000,C 0.000} C_DIS
LIN {X 268.406,Y 109.810,Z 138.306,A -157.750,B 90.000,C 0.000} C_DIS
LIN {X 268.505,Y 109.568,Z 138.105,A -157.801,B 90.000,C 0.000} C_DIS
LIN {X 269.307,Y 107.580,Z 136.819,A -158.225,B 90.000,C 0.000} C_DIS
LIN {X 269.349,Y 107.476,Z 136.739,A -158.247,B 90.000,C 0.000} C_DIS
LIN {X 269.485,Y 107.135,Z 136.508,A -158.319,B 90.000,C 0.000} C_DIS
LIN {X 269.506,Y 107.083,Z 136.455,A -158.331,B 90.000,C 0.000} C_DIS
LIN {X 269.672,Y 106.662,Z 136.206,A -158.420,B 90.000,C 0.000} C_DIS
LIN {X 269.763,Y 106.434,Z 136.022,A -158.468,B 90.000,C 0.000} C_DIS
LIN {X 269.926,Y 106.018,Z 135.773,A -158.557,B 90.000,C 0.000} C_DIS
LIN {X 270.007,Y 105.812,Z 135.602,A -158.601,B 90.000,C 0.000} C_DIS
LIN {X 270.324,Y 104.999,Z 135.047,A -158.773,B 90.000,C 0.000} C_DIS
LIN {X 270.382,Y 104.851,Z 134.976,A -158.804,B 90.000,C 0.000} C_DIS
LIN {X 270.438,Y 104.705,Z 134.805,A -158.835,B 90.000,C 0.000} C_DIS
LIN {X 270.568,Y 104.370,Z 134.518,A -158.906,B 90.000,C 0.000} C_DIS
LIN {X 270.784,Y 103.806,Z 133.620,A -159.025,B 90.000,C 0.000} C_DIS
LIN {X 270.788,Y 103.796,Z 133.549,A -159.028,B 90.000,C 0.000} C_DIS
LIN {X 270.880,Y 103.558,Z 132.964,A -159.078,B 90.000,C 0.000} C_DIS
LIN {X 270.931,Y 103.425,Z 132.865,A -159.106,B 90.000,C 0.000} C_DIS
LIN {X 270.913,Y 103.471,Z 132.991,A -159.096,B 90.000,C 0.000} C_DIS
LIN {X 270.901,Y 103.503,Z 133.358,A -159.090,B 90.000,C 0.000} C_DIS
LIN {X 270.858,Y 103.614,Z 133.667,A -159.066,B 90.000,C 0.000} C_DIS
LIN {X 270.834,Y 103.678,Z 134.028,A -159.053,B 90.000,C 0.000} C_DIS
LIN {X 270.738,Y 103.927,Z 134.577,A -159.000,B 90.000,C 0.000} C_DIS
LIN {X 270.721,Y 103.971,Z 134.620,A -158.991,B 90.000,C 0.000} C_DIS
LIN {X 270.709,Y 104.003,Z 134.777,A -158.984,B 90.000,C 0.000} C_DIS
LIN {X 270.671,Y 104.102,Z 135.061,A -158.963,B 90.000,C 0.000} C_DIS
LIN {X 270.595,Y 104.298,Z 135.463,A -158.921,B 90.000,C 0.000} C_DIS
LIN {X 270.574,Y 104.354,Z 135.545,A -158.909,B 90.000,C 0.000} C_DIS
LIN {X 270.556,Y 104.401,Z 135.659,A -158.900,B 90.000,C 0.000} C_DIS
LIN {X 270.534,Y 104.457,Z 135.735,A -158.888,B 90.000,C 0.000} C_DIS
LIN {X 270.145,Y 105.461,Z 137.299,A -158.675,B 90.000,C 0.000} C_DIS
LIN {X 270.090,Y 105.599,Z 137.422,A -158.646,B 90.000,C 0.000} C_DIS
LIN {X 270.060,Y 105.677,Z 137.508,A -158.629,B 90.000,C 0.000} C_DIS
LIN {X 270.038,Y 105.733,Z 137.593,A -158.617,B 90.000,C 0.000} C_DIS
LIN {X 270.028,Y 105.759,Z 137.646,A -158.612,B 90.000,C 0.000} C_DIS
LIN {X 269.967,Y 105.913,Z 137.825,A -158.579,B 90.000,C 0.000} C_DIS
LIN {X 269.954,Y 105.948,Z 137.877,A -158.572,B 90.000,C 0.000} C_DIS
LIN {X 269.496,Y 107.106,Z 138.863,A -158.326,B 90.000,C 0.000} C_DIS
LIN {X 269.406,Y 107.333,Z 138.980,A -158.277,B 90.000,C 0.000} C_DIS
LIN {X 269.138,Y 108.004,Z 139.491,A -158.135,B 90.000,C 0.000} C_DIS
LIN {X 270.059,Y 105.681,Z 139.531,A -158.628,B 90.000,C 0.000} C_DIS
LIN {X 270.958,Y 103.352,Z 139.667,A -159.122,B 90.000,C 0.000} C_DIS
LIN {X 271.710,Y 101.359,Z 139.836,A -159.542,B 90.000,C 0.000} C_DIS
LIN {X 271.765,Y 101.212,Z 139.872,A -159.573,B 90.000,C 0.000} C_DIS
LIN {X 272.037,Y 100.479,Z 139.945,A -159.728,B 90.000,C 0.000} C_DIS
LIN {X 272.118,Y 100.259,Z 140.016,A -159.774,B 90.000,C 0.000} C_DIS
LIN {X 272.455,Y 99.339,Z 140.122,A -159.968,B 90.000,C 0.000} C_DIS
LIN {X 272.473,Y 99.290,Z 140.151,A -159.978,B 90.000,C 0.000} C_DIS
LIN {X 272.570,Y 99.023,Z 140.190,A -160.034,B 90.000,C 0.000} C_DIS
LIN {X 273.340,Y 96.877,Z 140.786,A -160.485,B 90.000,C 0.000} C_DIS
LIN {X 273.360,Y 96.821,Z 140.837,A -160.496,B 90.000,C 0.000} C_DIS
LIN {X 273.485,Y 96.469,Z 140.950,A -160.570,B 90.000,C 0.000} C_DIS
LIN {X 273.749,Y 95.715,Z 141.459,A -160.728,B 90.000,C 0.000} C_DIS
LIN {X 273.787,Y 95.607,Z 141.482,A -160.751,B 90.000,C 0.000} C_DIS
LIN {X 274.531,Y 93.448,Z 140.465,A -161.202,B 90.000,C 0.000} C_DIS
LIN {X 274.802,Y 92.650,Z 139.983,A -161.368,B 90.000,C 0.000} C_DIS
LIN {X 274.958,Y 92.185,Z 139.627,A -161.465,B 90.000,C 0.000} C_DIS
LIN {X 275.204,Y 91.448,Z 138.868,A -161.619,B 90.000,C 0.000} C_DIS
LIN {X 275.276,Y 91.230,Z 138.466,A -161.664,B 90.000,C 0.000} C_DIS
LIN {X 275.295,Y 91.173,Z 138.390,A -161.676,B 90.000,C 0.000} C_DIS
LIN {X 275.311,Y 91.125,Z 138.276,A -161.686,B 90.000,C 0.000} C_DIS
LIN {X 275.347,Y 91.018,Z 138.105,A -161.708,B 90.000,C 0.000} C_DIS
LIN {X 275.397,Y 90.865,Z 138.575,A -161.740,B 90.000,C 0.000} C_DIS
LIN {X 275.419,Y 90.800,Z 139.091,A -161.754,B 90.000,C 0.000} C_DIS
LIN {X 275.424,Y 90.785,Z 139.552,A -161.757,B 90.000,C 0.000} C_DIS
LIN {X 275.393,Y 90.879,Z 140.333,A -161.737,B 90.000,C 0.000} C_DIS
LIN {X 273.493,Y 90.252,Z 140.333,A -161.737,B 90.000,C 0.000} C_DIS
WAIT SEC 0.1
RET=EKI_SetBool("oxy","torchState",FALSE)
RET = EKI_Send("oxy","torchState")
LIN {X 256.400,Y 84.611,Z 140.333,A -161.737,B 90.000,C 0.000} C_DIS
LIN {X 252.721,Y 95.037,Z 126.043,A -159.391,B 90.000,C 0.000} C_DIS
LIN {X 269.569,Y 101.372,Z 126.043,A -159.391,B 90.000,C 0.000} C_DIS
LIN {X 271.441,Y 102.076,Z 126.043,A -159.391,B 90.000,C 0.000} C_DIS
WAIT SEC 1
RET=EKI_SetBool("oxy","torchState",TRUE)
RET = EKI_Send("oxy","torchState")
LIN {X 270.669,Y 104.108,Z 127.277,A -158.962,B 90.000,C 0.000} C_DIS
LIN {X 270.498,Y 104.552,Z 127.448,A -158.868,B 90.000,C 0.000} C_DIS
LIN {X 270.210,Y 105.293,Z 127.547,A -158.711,B 90.000,C 0.000} C_DIS
LIN {X 270.039,Y 105.730,Z 127.523,A -158.618,B 90.000,C 0.000} C_DIS
LIN {X 269.748,Y 106.471,Z 127.232,A -158.461,B 90.000,C 0.000} C_DIS
LIN {X 269.667,Y 106.675,Z 127.195,A -158.417,B 90.000,C 0.000} C_DIS
LIN {X 269.356,Y 107.458,Z 126.896,A -158.251,B 90.000,C 0.000} C_DIS
LIN {X 269.328,Y 107.529,Z 126.849,A -158.236,B 90.000,C 0.000} C_DIS
LIN {X 269.074,Y 108.163,Z 126.556,A -158.101,B 90.000,C 0.000} C_DIS
LIN {X 268.992,Y 108.366,Z 126.519,A -158.058,B 90.000,C 0.000} C_DIS
LIN {X 268.476,Y 109.639,Z 125.925,A -157.786,B 90.000,C 0.000} C_DIS
LIN {X 268.390,Y 109.850,Z 125.878,A -157.741,B 90.000,C 0.000} C_DIS
LIN {X 268.183,Y 110.355,Z 125.635,A -157.633,B 90.000,C 0.000} C_DIS
LIN {X 268.145,Y 110.447,Z 125.626,A -157.614,B 90.000,C 0.000} C_DIS
LIN {X 267.264,Y 112.561,Z 124.625,A -157.161,B 90.000,C 0.000} C_DIS
LIN {X 266.834,Y 113.577,Z 124.102,A -156.943,B 90.000,C 0.000} C_DIS
LIN {X 266.783,Y 113.695,Z 124.083,A -156.918,B 90.000,C 0.000} C_DIS
LIN {X 266.724,Y 113.835,Z 124.020,A -156.888,B 90.000,C 0.000} C_DIS
LIN {X 266.696,Y 113.900,Z 124.009,A -156.874,B 90.000,C 0.000} C_DIS
LIN {X 266.335,Y 114.741,Z 123.586,A -156.693,B 90.000,C 0.000} C_DIS
LIN {X 266.318,Y 114.780,Z 123.539,A -156.684,B 90.000,C 0.000} C_DIS
LIN {X 266.286,Y 114.855,Z 123.483,A -156.668,B 90.000,C 0.000} C_DIS
LIN {X 266.183,Y 115.094,Z 123.339,A -156.617,B 90.000,C 0.000} C_DIS
LIN {X 266.042,Y 115.419,Z 123.198,A -156.547,B 90.000,C 0.000} C_DIS
LIN {X 266.002,Y 115.512,Z 123.141,A -156.527,B 90.000,C 0.000} C_DIS
LIN {X 265.974,Y 115.577,Z 123.084,A -156.513,B 90.000,C 0.000} C_DIS
LIN {X 265.684,Y 116.242,Z 122.720,A -156.370,B 90.000,C 0.000} C_DIS
LIN {X 265.579,Y 116.480,Z 122.572,A -156.318,B 90.000,C 0.000} C_DIS
LIN {X 265.432,Y 116.815,Z 122.335,A -156.246,B 90.000,C 0.000} C_DIS
LIN {X 265.386,Y 116.919,Z 122.291,A -156.224,B 90.000,C 0.000} C_DIS
LIN {X 265.318,Y 117.075,Z 122.171,A -156.190,B 90.000,C 0.000} C_DIS
LIN {X 265.272,Y 117.179,Z 122.120,A -156.167,B 90.000,C 0.000} C_DIS
LIN {X 265.275,Y 117.172,Z 122.075,A -156.169,B 90.000,C 0.000} C_DIS
LIN {X 265.334,Y 117.037,Z 122.052,A -156.198,B 90.000,C 0.000} C_DIS
LIN {X 266.330,Y 114.745,Z 121.990,A -156.692,B 90.000,C 0.000} C_DIS
LIN {X 267.310,Y 112.449,Z 121.851,A -157.185,B 90.000,C 0.000} C_DIS
LIN {X 268.254,Y 110.177,Z 121.408,A -157.671,B 90.000,C 0.000} C_DIS
LIN {X 269.160,Y 107.944,Z 120.743,A -158.147,B 90.000,C 0.000} C_DIS
LIN {X 270.009,Y 105.808,Z 119.760,A -158.601,B 90.000,C 0.000} C_DIS
LIN {X 270.164,Y 105.412,Z 119.554,A -158.685,B 90.000,C 0.000} C_DIS
LIN {X 270.336,Y 104.969,Z 119.215,A -158.779,B 90.000,C 0.000} C_DIS
LIN {X 270.407,Y 104.786,Z 119.116,A -158.818,B 90.000,C 0.000} C_DIS
LIN {X 270.569,Y 104.367,Z 118.817,A -158.907,B 90.000,C 0.000} C_DIS
LIN {X 270.626,Y 104.218,Z 118.646,A -158.938,B 90.000,C 0.000} C_DIS
LIN {X 270.657,Y 104.139,Z 118.588,A -158.955,B 90.000,C 0.000} C_DIS
LIN {X 270.978,Y 103.300,Z 117.778,A -159.133,B 90.000,C 0.000} C_DIS
LIN {X 271.441,Y 102.078,Z 116.038,A -159.391,B 90.000,C 0.000} C_DIS
LIN {X 271.546,Y 101.798,Z 115.536,A -159.450,B 90.000,C 0.000} C_DIS
LIN {X 271.567,Y 101.742,Z 115.460,A -159.462,B 90.000,C 0.000} C_DIS
LIN {X 271.585,Y 101.695,Z 115.346,A -159.472,B 90.000,C 0.000} C_DIS
LIN {X 271.606,Y 101.639,Z 115.265,A -159.483,B 90.000,C 0.000} C_DIS
LIN {X 271.654,Y 101.508,Z 115.005,A -159.511,B 90.000,C 0.000} C_DIS
LIN {X 271.659,Y 101.495,Z 114.934,A -159.514,B 90.000,C 0.000} C_DIS
LIN {X 271.748,Y 101.259,Z 114.379,A -159.564,B 90.000,C 0.000} C_DIS
LIN {X 271.751,Y 101.248,Z 114.288,A -159.566,B 90.000,C 0.000} C_DIS
LIN {X 271.792,Y 101.138,Z 113.930,A -159.589,B 90.000,C 0.000} C_DIS
LIN {X 271.853,Y 100.976,Z 113.064,A -159.623,B 90.000,C 0.000} C_DIS
LIN {X 271.859,Y 100.958,Z 113.014,A -159.627,B 90.000,C 0.000} C_DIS
LIN {X 271.885,Y 100.888,Z 112.388,A -159.642,B 90.000,C 0.000} C_DIS
LIN {X 271.858,Y 100.963,Z 109.889,A -159.626,B 90.000,C 0.000} C_DIS
LIN {X 271.857,Y 100.965,Z 109.856,A -159.625,B 90.000,C 0.000} C_DIS
LIN {X 271.648,Y 101.526,Z 107.609,A -159.507,B 90.000,C 0.000} C_DIS
LIN {X 271.547,Y 101.796,Z 106.983,A -159.450,B 90.000,C 0.000} C_DIS
LIN {X 271.467,Y 102.009,Z 106.571,A -159.405,B 90.000,C 0.000} C_DIS
LIN {X 271.366,Y 102.278,Z 106.149,A -159.349,B 90.000,C 0.000} C_DIS
LIN {X 271.335,Y 102.358,Z 106.072,A -159.332,B 90.000,C 0.000} C_DIS
LIN {X 271.305,Y 102.437,Z 106.015,A -159.315,B 90.000,C 0.000} C_DIS
LIN {X 271.143,Y 102.865,Z 105.521,A -159.224,B 90.000,C 0.000} C_DIS
LIN {X 270.950,Y 103.374,Z 105.105,A -159.117,B 90.000,C 0.000} C_DIS
LIN {X 270.922,Y 103.448,Z 105.062,A -159.101,B 90.000,C 0.000} C_DIS
LIN {X 270.716,Y 103.986,Z 104.618,A -158.987,B 90.000,C 0.000} C_DIS
LIN {X 270.737,Y 103.930,Z 102.119,A -158.999,B 90.000,C 0.000} C_DIS
LIN {X 270.759,Y 103.874,Z 99.620,A -159.011,B 90.000,C 0.000} C_DIS
LIN {X 270.789,Y 103.795,Z 97.121,A -159.028,B 90.000,C 0.000} C_DIS
LIN {X 270.820,Y 103.714,Z 94.623,A -159.045,B 90.000,C 0.000} C_DIS
LIN {X 270.843,Y 103.654,Z 92.124,A -159.058,B 90.000,C 0.000} C_DIS
LIN {X 270.842,Y 103.656,Z 90.592,A -159.057,B 90.000,C 0.000} C_DIS
LIN {X 270.796,Y 103.777,Z 90.255,A -159.032,B 90.000,C 0.000} C_DIS
LIN {X 270.307,Y 105.044,Z 88.157,A -158.763,B 90.000,C 0.000} C_DIS
LIN {X 269.880,Y 106.135,Z 85.948,A -158.532,B 90.000,C 0.000} C_DIS
LIN {X 269.527,Y 107.029,Z 83.640,A -158.342,B 90.000,C 0.000} C_DIS
LIN {X 269.249,Y 107.725,Z 81.256,A -158.194,B 90.000,C 0.000} C_DIS
LIN {X 269.030,Y 108.271,Z 78.826,A -158.078,B 90.000,C 0.000} C_DIS
LIN {X 268.898,Y 108.599,Z 76.351,A -158.008,B 90.000,C 0.000} C_DIS
LIN {X 268.867,Y 108.677,Z 73.853,A -157.991,B 90.000,C 0.000} C_DIS
LIN {X 268.879,Y 108.646,Z 71.353,A -157.998,B 90.000,C 0.000} C_DIS
LIN {X 268.906,Y 108.579,Z 70.569,A -158.012,B 90.000,C 0.000} C_DIS
LIN {X 268.999,Y 108.350,Z 68.630,A -158.061,B 90.000,C 0.000} C_DIS
LIN {X 269.007,Y 108.330,Z 68.578,A -158.065,B 90.000,C 0.000} C_DIS
LIN {X 269.219,Y 107.802,Z 66.144,A -158.178,B 90.000,C 0.000} C_DIS
LIN {X 269.370,Y 107.424,Z 64.681,A -158.258,B 90.000,C 0.000} C_DIS
LIN {X 269.381,Y 107.395,Z 64.538,A -158.264,B 90.000,C 0.000} C_DIS
LIN {X 269.704,Y 106.582,Z 62.196,A -158.437,B 90.000,C 0.000} C_DIS
LIN {X 270.076,Y 105.637,Z 59.912,A -158.638,B 90.000,C 0.000} C_DIS
LIN {X 270.185,Y 105.356,Z 59.361,A -158.697,B 90.000,C 0.000} C_DIS
LIN {X 270.251,Y 105.187,Z 58.891,A -158.733,B 90.000,C 0.000} C_DIS
LIN {X 270.265,Y 105.150,Z 58.849,A -158.741,B 90.000,C 0.000} C_DIS
LIN {X 270.299,Y 105.064,Z 58.723,A -158.759,B 90.000,C 0.000} C_DIS
LIN {X 270.341,Y 104.956,Z 58.519,A -158.782,B 90.000,C 0.000} C_DIS
LIN {X 270.377,Y 104.862,Z 58.537,A -158.802,B 90.000,C 0.000} C_DIS
LIN {X 270.350,Y 104.933,Z 58.876,A -158.787,B 90.000,C 0.000} C_DIS
LIN {X 270.339,Y 104.961,Z 58.963,A -158.781,B 90.000,C 0.000} C_DIS
LIN {X 270.295,Y 105.074,Z 59.904,A -158.757,B 90.000,C 0.000} C_DIS
LIN {X 270.273,Y 105.132,Z 60.060,A -158.745,B 90.000,C 0.000} C_DIS
LIN {X 270.171,Y 105.393,Z 62.544,A -158.689,B 90.000,C 0.000} C_DIS
LIN {X 270.163,Y 105.414,Z 62.661,A -158.685,B 90.000,C 0.000} C_DIS
LIN {X 270.101,Y 105.572,Z 65.155,A -158.651,B 90.000,C 0.000} C_DIS
LIN {X 270.096,Y 105.584,Z 67.655,A -158.649,B 90.000,C 0.000} C_DIS
LIN {X 270.126,Y 105.507,Z 70.153,A -158.665,B 90.000,C 0.000} C_DIS
LIN {X 270.213,Y 105.285,Z 72.642,A -158.712,B 90.000,C 0.000} C_DIS
LIN {X 270.367,Y 104.888,Z 75.105,A -158.796,B 90.000,C 0.000} C_DIS
LIN {X 270.582,Y 104.334,Z 77.534,A -158.914,B 90.000,C 0.000} C_DIS
LIN {X 270.807,Y 103.749,Z 79.401,A -159.038,B 90.000,C 0.000} C_DIS
LIN {X 270.812,Y 103.735,Z 79.489,A -159.041,B 90.000,C 0.000} C_DIS
LIN {X 271.171,Y 102.794,Z 81.775,A -159.240,B 90.000,C 0.000} C_DIS
LIN {X 271.387,Y 102.221,Z 82.973,A -159.361,B 90.000,C 0.000} C_DIS
LIN {X 271.623,Y 101.591,Z 84.055,A -159.494,B 90.000,C 0.000} C_DIS
LIN {X 272.143,Y 100.191,Z 86.060,A -159.789,B 90.000,C 0.000} C_DIS
LIN {X 272.159,Y 100.147,Z 86.124,A -159.798,B 90.000,C 0.000} C_DIS
LIN {X 272.756,Y 98.506,Z 87.913,A -160.143,B 90.000,C 0.000} C_DIS
LIN {X 272.923,Y 98.046,Z 88.390,A -160.239,B 90.000,C 0.000} C_DIS
LIN {X 273.061,Y 97.661,Z 88.936,A -160.320,B 90.000,C 0.000} C_DIS
LIN {X 273.092,Y 97.574,Z 89.029,A -160.339,B 90.000,C 0.000} C_DIS
LIN {X 273.110,Y 97.524,Z 89.048,A -160.349,B 90.000,C 0.000} C_DIS
LIN {X 273.143,Y 97.430,Z 89.217,A -160.369,B 90.000,C 0.000} C_DIS
LIN {X 273.397,Y 96.718,Z 90.242,A -160.518,B 90.000,C 0.000} C_DIS
LIN {X 273.437,Y 96.604,Z 90.484,A -160.542,B 90.000,C 0.000} C_DIS
LIN {X 273.824,Y 95.500,Z 92.693,A -160.773,B 90.000,C 0.000} C_DIS
LIN {X 274.106,Y 94.689,Z 95.041,A -160.943,B 90.000,C 0.000} C_DIS
LIN {X 274.287,Y 94.163,Z 97.478,A -161.053,B 90.000,C 0.000} C_DIS
LIN {X 274.387,Y 93.871,Z 99.959,A -161.114,B 90.000,C 0.000} C_DIS
LIN {X 274.421,Y 93.771,Z 102.457,A -161.134,B 90.000,C 0.000} C_DIS
LIN {X 274.402,Y 93.828,Z 104.956,A -161.123,B 90.000,C 0.000} C_DIS
LIN {X 274.327,Y 94.046,Z 107.445,A -161.077,B 90.000,C 0.000} C_DIS
LIN {X 274.270,Y 94.214,Z 108.733,A -161.042,B 90.000,C 0.000} C_DIS
LIN {X 274.259,Y 94.245,Z 108.860,A -161.035,B 90.000,C 0.000} C_DIS
LIN {X 274.248,Y 94.277,Z 108.914,A -161.029,B 90.000,C 0.000} C_DIS
LIN {X 274.175,Y 94.489,Z 110.285,A -160.984,B 90.000,C 0.000} C_DIS
LIN {X 274.164,Y 94.521,Z 110.340,A -160.978,B 90.000,C 0.000} C_DIS
LIN {X 274.152,Y 94.556,Z 110.453,A -160.971,B 90.000,C 0.000} C_DIS
LIN {X 274.141,Y 94.587,Z 110.738,A -160.964,B 90.000,C 0.000} C_DIS
LIN {X 274.129,Y 94.622,Z 110.852,A -160.957,B 90.000,C 0.000} C_DIS
LIN {X 274.118,Y 94.653,Z 110.908,A -160.950,B 90.000,C 0.000} C_DIS
LIN {X 273.941,Y 95.164,Z 113.127,A -160.843,B 90.000,C 0.000} C_DIS
LIN {X 273.936,Y 95.178,Z 113.241,A -160.840,B 90.000,C 0.000} C_DIS
LIN {X 273.872,Y 95.362,Z 113.867,A -160.802,B 90.000,C 0.000} C_DIS
LIN {X 273.868,Y 95.374,Z 113.981,A -160.800,B 90.000,C 0.000} C_DIS
LIN {X 273.617,Y 96.092,Z 116.095,A -160.649,B 90.000,C 0.000} C_DIS
LIN {X 273.605,Y 96.125,Z 116.314,A -160.642,B 90.000,C 0.000} C_DIS
LIN {X 273.277,Y 97.055,Z 118.611,A -160.447,B 90.000,C 0.000} C_DIS
LIN {X 273.206,Y 97.256,Z 119.077,A -160.405,B 90.000,C 0.000} C_DIS
LIN {X 273.185,Y 97.313,Z 119.158,A -160.393,B 90.000,C 0.000} C_DIS
LIN {X 273.099,Y 97.554,Z 119.723,A -160.343,B 90.000,C 0.000} C_DIS
LIN {X 273.096,Y 97.564,Z 119.794,A -160.341,B 90.000,C 0.000} C_DIS
LIN {X 272.918,Y 98.060,Z 120.727,A -160.237,B 90.000,C 0.000} C_DIS
LIN {X 272.898,Y 98.116,Z 120.808,A -160.225,B 90.000,C 0.000} C_DIS
LIN {X 272.881,Y 98.164,Z 120.922,A -160.215,B 90.000,C 0.000} C_DIS
LIN {X 272.860,Y 98.220,Z 120.999,A -160.203,B 90.000,C 0.000} C_DIS
LIN {X 272.783,Y 98.434,Z 121.415,A -160.158,B 90.000,C 0.000} C_DIS
LIN {X 272.703,Y 98.657,Z 121.776,A -160.111,B 90.000,C 0.000} C_DIS
LIN {X 272.688,Y 98.699,Z 121.889,A -160.102,B 90.000,C 0.000} C_DIS
LIN {X 272.635,Y 98.845,Z 122.097,A -160.072,B 90.000,C 0.000} C_DIS
LIN {X 272.124,Y 100.243,Z 124.106,A -159.777,B 90.000,C 0.000} C_DIS
LIN {X 271.909,Y 100.825,Z 124.848,A -159.655,B 90.000,C 0.000} C_DIS
LIN {X 271.441,Y 102.076,Z 126.043,A -159.391,B 90.000,C 0.000} C_DIS
LIN {X 269.569,Y 101.372,Z 126.043,A -159.391,B 90.000,C 0.000} C_DIS
WAIT SEC 0.1
RET=EKI_SetBool("oxy","torchState",FALSE)
RET = EKI_Send("oxy","torchState")
LIN {X 252.721,Y 95.037,Z 126.043,A -159.391,B 90.000,C 0.000} C_DIS
LIN {X 247.690,Y 107.468,Z 129.506,A -156.545,B 90.000,C 0.000} C_DIS
LIN {X 264.203,Y 114.633,Z 129.506,A -156.545,B 90.000,C 0.000} C_DIS
LIN {X 266.038,Y 115.429,Z 129.506,A -156.545,B 90.000,C 0.000} C_DIS
WAIT SEC 1
RET=EKI_SetBool("oxy","torchState",TRUE)
RET = EKI_Send("oxy","torchState")
LIN {X 266.150,Y 115.170,Z 131.989,A -156.601,B 90.000,C 0.000} C_DIS
LIN {X 266.153,Y 115.164,Z 133.769,A -156.602,B 90.000,C 0.000} C_DIS
LIN {X 266.102,Y 115.280,Z 134.492,A -156.577,B 90.000,C 0.000} C_DIS
LIN {X 266.042,Y 115.419,Z 134.862,A -156.547,B 90.000,C 0.000} C_DIS
LIN {X 266.028,Y 115.451,Z 134.975,A -156.540,B 90.000,C 0.000} C_DIS
LIN {X 265.834,Y 115.897,Z 135.783,A -156.444,B 90.000,C 0.000} C_DIS
LIN {X 265.750,Y 116.090,Z 135.952,A -156.402,B 90.000,C 0.000} C_DIS
LIN {X 265.133,Y 117.492,Z 137.657,A -156.100,B 90.000,C 0.000} C_DIS
LIN {X 265.099,Y 117.570,Z 137.706,A -156.083,B 90.000,C 0.000} C_DIS
LIN {X 265.029,Y 117.727,Z 137.877,A -156.049,B 90.000,C 0.000} C_DIS
LIN {X 264.935,Y 117.939,Z 138.048,A -156.003,B 90.000,C 0.000} C_DIS
LIN {X 264.801,Y 118.240,Z 138.389,A -155.938,B 90.000,C 0.000} C_DIS
LIN {X 264.706,Y 118.452,Z 138.560,A -155.892,B 90.000,C 0.000} C_DIS
LIN {X 264.670,Y 118.531,Z 138.645,A -155.875,B 90.000,C 0.000} C_DIS
LIN {X 264.641,Y 118.596,Z 138.733,A -155.861,B 90.000,C 0.000} C_DIS
LIN {X 264.468,Y 118.983,Z 139.072,A -155.777,B 90.000,C 0.000} C_DIS
LIN {X 264.405,Y 119.122,Z 139.243,A -155.747,B 90.000,C 0.000} C_DIS
LIN {X 264.359,Y 119.225,Z 139.328,A -155.725,B 90.000,C 0.000} C_DIS
LIN {X 264.322,Y 119.305,Z 139.413,A -155.707,B 90.000,C 0.000} C_DIS
LIN {X 263.872,Y 120.297,Z 140.338,A -155.492,B 90.000,C 0.000} C_DIS
LIN {X 263.808,Y 120.439,Z 140.437,A -155.461,B 90.000,C 0.000} C_DIS
LIN {X 263.560,Y 120.981,Z 140.950,A -155.344,B 90.000,C 0.000} C_DIS
LIN {X 263.497,Y 121.117,Z 141.034,A -155.314,B 90.000,C 0.000} C_DIS
LIN {X 263.068,Y 122.046,Z 141.860,A -155.112,B 90.000,C 0.000} C_DIS
LIN {X 262.704,Y 122.829,Z 142.543,A -154.941,B 90.000,C 0.000} C_DIS
LIN {X 262.604,Y 123.041,Z 142.745,A -154.895,B 90.000,C 0.000} C_DIS
LIN {X 262.281,Y 123.729,Z 143.183,A -154.745,B 90.000,C 0.000} C_DIS
LIN {X 262.011,Y 124.299,Z 143.337,A -154.620,B 90.000,C 0.000} C_DIS
LIN {X 261.543,Y 125.281,Z 143.318,A -154.405,B 90.000,C 0.000} C_DIS
LIN {X 261.488,Y 125.396,Z 143.262,A -154.380,B 90.000,C 0.000} C_DIS
LIN {X 261.315,Y 125.755,Z 143.209,A -154.301,B 90.000,C 0.000} C_DIS
LIN {X 261.218,Y 125.956,Z 143.139,A -154.257,B 90.000,C 0.000} C_DIS
LIN {X 261.155,Y 126.088,Z 143.113,A -154.228,B 90.000,C 0.000} C_DIS
LIN {X 261.116,Y 126.169,Z 143.086,A -154.211,B 90.000,C 0.000} C_DIS
LIN {X 261.093,Y 126.216,Z 143.061,A -154.200,B 90.000,C 0.000} C_DIS
LIN {X 260.994,Y 126.421,Z 142.999,A -154.155,B 90.000,C 0.000} C_DIS
LIN {X 260.918,Y 126.578,Z 142.912,A -154.121,B 90.000,C 0.000} C_DIS
LIN {X 260.492,Y 127.452,Z 142.144,A -153.929,B 90.000,C 0.000} C_DIS
LIN {X 260.471,Y 127.496,Z 142.059,A -153.919,B 90.000,C 0.000} C_DIS
LIN {X 260.364,Y 127.713,Z 141.803,A -153.871,B 90.000,C 0.000} C_DIS
LIN {X 260.216,Y 128.013,Z 141.495,A -153.805,B 90.000,C 0.000} C_DIS
LIN {X 260.182,Y 128.083,Z 141.405,A -153.790,B 90.000,C 0.000} C_DIS
LIN {X 260.143,Y 128.163,Z 141.322,A -153.772,B 90.000,C 0.000} C_DIS
LIN {X 260.119,Y 128.210,Z 141.292,A -153.762,B 90.000,C 0.000} C_DIS
LIN {X 259.513,Y 129.434,Z 139.751,A -153.492,B 90.000,C 0.000} C_DIS
LIN {X 259.462,Y 129.536,Z 139.707,A -153.469,B 90.000,C 0.000} C_DIS
LIN {X 259.054,Y 130.350,Z 138.608,A -153.290,B 90.000,C 0.000} C_DIS
LIN {X 259.003,Y 130.451,Z 138.567,A -153.267,B 90.000,C 0.000} C_DIS
LIN {X 258.614,Y 131.221,Z 137.534,A -153.097,B 90.000,C 0.000} C_DIS
LIN {X 258.437,Y 131.568,Z 136.994,A -153.020,B 90.000,C 0.000} C_DIS
LIN {X 258.373,Y 131.694,Z 136.854,A -152.992,B 90.000,C 0.000} C_DIS
LIN {X 257.763,Y 132.884,Z 134.963,A -152.728,B 90.000,C 0.000} C_DIS
LIN {X 257.214,Y 133.944,Z 132.766,A -152.492,B 90.000,C 0.000} C_DIS
LIN {X 257.087,Y 134.187,Z 132.081,A -152.438,B 90.000,C 0.000} C_DIS
LIN {X 257.029,Y 134.299,Z 131.391,A -152.413,B 90.000,C 0.000} C_DIS
LIN {X 257.037,Y 134.282,Z 130.595,A -152.416,B 90.000,C 0.000} C_DIS
LIN {X 257.121,Y 134.123,Z 129.604,A -152.452,B 90.000,C 0.000} C_DIS
LIN {X 257.265,Y 133.846,Z 128.546,A -152.514,B 90.000,C 0.000} C_DIS
LIN {X 257.397,Y 133.592,Z 128.059,A -152.570,B 90.000,C 0.000} C_DIS
LIN {X 257.425,Y 133.538,Z 127.977,A -152.582,B 90.000,C 0.000} C_DIS
LIN {X 257.448,Y 133.494,Z 127.863,A -152.592,B 90.000,C 0.000} C_DIS
LIN {X 257.503,Y 133.387,Z 127.693,A -152.616,B 90.000,C 0.000} C_DIS
LIN {X 257.516,Y 133.362,Z 127.640,A -152.621,B 90.000,C 0.000} C_DIS
LIN {X 257.556,Y 133.286,Z 127.549,A -152.638,B 90.000,C 0.000} C_DIS
LIN {X 257.597,Y 133.206,Z 127.482,A -152.656,B 90.000,C 0.000} C_DIS
LIN {X 257.772,Y 132.867,Z 127.067,A -152.731,B 90.000,C 0.000} C_DIS
LIN {X 258.055,Y 132.316,Z 126.674,A -152.854,B 90.000,C 0.000} C_DIS
LIN {X 258.253,Y 131.930,Z 126.665,A -152.939,B 90.000,C 0.000} C_DIS
LIN {X 258.414,Y 131.613,Z 126.846,A -153.010,B 90.000,C 0.000} C_DIS
LIN {X 258.581,Y 131.285,Z 127.845,A -153.083,B 90.000,C 0.000} C_DIS
LIN {X 258.753,Y 130.947,Z 128.389,A -153.157,B 90.000,C 0.000} C_DIS
LIN {X 258.896,Y 130.663,Z 128.660,A -153.220,B 90.000,C 0.000} C_DIS
LIN {X 258.958,Y 130.540,Z 128.740,A -153.248,B 90.000,C 0.000} C_DIS
LIN {X 259.191,Y 130.076,Z 128.934,A -153.350,B 90.000,C 0.000} C_DIS
LIN {X 259.507,Y 129.446,Z 129.051,A -153.489,B 90.000,C 0.000} C_DIS
LIN {X 259.622,Y 129.215,Z 129.033,A -153.540,B 90.000,C 0.000} C_DIS
LIN {X 259.761,Y 128.936,Z 128.831,A -153.602,B 90.000,C 0.000} C_DIS
LIN {X 259.780,Y 128.896,Z 128.779,A -153.611,B 90.000,C 0.000} C_DIS
LIN {X 260.742,Y 126.940,Z 127.555,A -154.041,B 90.000,C 0.000} C_DIS
LIN {X 261.672,Y 125.011,Z 126.962,A -154.464,B 90.000,C 0.000} C_DIS
LIN {X 261.732,Y 124.886,Z 126.891,A -154.492,B 90.000,C 0.000} C_DIS
LIN {X 261.792,Y 124.759,Z 124.395,A -154.520,B 90.000,C 0.000} C_DIS
LIN {X 261.820,Y 124.701,Z 121.896,A -154.532,B 90.000,C 0.000} C_DIS
LIN {X 261.848,Y 124.642,Z 119.397,A -154.545,B 90.000,C 0.000} C_DIS
LIN {X 261.882,Y 124.571,Z 116.898,A -154.561,B 90.000,C 0.000} C_DIS
LIN {X 261.911,Y 124.509,Z 114.399,A -154.574,B 90.000,C 0.000} C_DIS
LIN {X 261.937,Y 124.455,Z 113.378,A -154.586,B 90.000,C 0.000} C_DIS
LIN {X 261.903,Y 124.526,Z 113.314,A -154.570,B 90.000,C 0.000} C_DIS
LIN {X 260.831,Y 126.755,Z 113.677,A -154.082,B 90.000,C 0.000} C_DIS
LIN {X 259.738,Y 128.980,Z 114.003,A -153.592,B 90.000,C 0.000} C_DIS
LIN {X 259.717,Y 129.023,Z 114.007,A -153.583,B 90.000,C 0.000} C_DIS
LIN {X 259.690,Y 129.077,Z 113.992,A -153.571,B 90.000,C 0.000} C_DIS
LIN {X 258.567,Y 131.311,Z 113.978,A -153.077,B 90.000,C 0.000} C_DIS
